LIN {X 0,Y 530.487,Z 752.804,A -85,B 0,C 180,E1 -4231.898,E2 -4231.898} C_VEL
LIN {X 0,Y 530.55,Z 749.173,A -85,B 0,C 180,E1 -4233.037,E2 -4233.037} C_VEL
LIN {X 0,Y 530.595,Z 744.443,A -85,B 0,C 180,E1 -4234.178,E2 -4234.178} C_VEL
LIN {X 0,Y 530.684,Z 738.476,A -85,B 0,C 180,E1 -4235.319,E2 -4235.319} C_VEL
LIN {X 0,Y 530.899,Z 731.608,A -85,B 0,C 180,E1 -4236.382,E2 -4236.382} C_VEL
LIN {X 0,Y 531.003,Z 723.637,A -85,B 0,C 180,E1 -4237.395,E2 -4237.395} C_VEL
LIN {X 0,Y 531.252,Z 713.214,A -85,B 0,C 180,E1 -4238.463,E2 -4238.463} C_VEL
LIN {X 0,Y 531.557,Z 702.842,A -85,B 0,C 180,E1 -4239.321,E2 -4239.321} C_VEL
LIN {X 0,Y 531.809,Z 691.176,A -85,B 0,C 180,E1 -4240.084,E2 -4240.084} C_VEL
LIN {X 0,Y 532.085,Z 678.914,A -85,B 0,C 180,E1 -4240.704,E2 -4240.704} C_VEL
LIN {X 0,Y 532.25,Z 666.678,A -85,B 0,C 180,E1 -4241.158,E2 -4241.158} C_VEL
LIN {X 0,Y 532.378,Z 652.951,A -85,B 0,C 180,E1 -4241.493,E2 -4241.493} C_VEL
LIN {X 0,Y 532.801,Z 555.086,A -85,B 0,C 180,E1 -4242.828,E2 -4242.828} C_VEL
LIN {X 0,Y 531.345,Z 546.226,A -85,B 0,C 180,E1 -4242.994,E2 -4242.994} C_VEL
LIN {X 0,Y 531.703,Z 526.604,A -85,B 0,C 180,E1 -4246.115,E2 -4246.115} C_VEL
LIN {X 0,Y 532.063,Z 506.634,A -85,B 0,C 180,E1 -4249.282,E2 -4249.282} C_VEL
LIN {X 0,Y 532.005,Z 498.624,A -85,B 0,C 180,E1 -4250.561,E2 -4250.561} C_VEL
LIN {X 0,Y 531.024,Z 493.342,A -85,B 0,C 180,E1 -4251.445,E2 -4251.445} C_VEL
LIN {X 0,Y 530.974,Z 493.345,A -85,B 0,C 180,E1 -4254.224,E2 -4254.224} C_VEL
LIN {X 0,Y 531.004,Z 493.343,A -85,B 0,C 180,E1 -4256.743,E2 -4256.743} C_VEL
LIN {X 0,Y 530.984,Z 493.345,A -85,B 0,C 180,E1 -4259.322,E2 -4259.322} C_VEL
LIN {X 0,Y 530.981,Z 493.34,A -85,B 0,C 180,E1 -4262.102,E2 -4262.102} C_VEL
LIN {X 0,Y 530.977,Z 493.347,A -85,B 0,C 180,E1 -4264.851,E2 -4264.851} C_VEL
LIN {X 0,Y 530.966,Z 493.343,A -85,B 0,C 180,E1 -4267.507,E2 -4267.507} C_VEL
LIN {X 0,Y 530.984,Z 493.34,A -85,B 0,C 180,E1 -4270.431,E2 -4270.431} C_VEL
LIN {X 0,Y 530.97,Z 493.343,A -85,B 0,C 180,E1 -4273.281,E2 -4273.281} C_VEL
LIN {X 0,Y 530.985,Z 493.336,A -85,B 0,C 180,E1 -4275.62,E2 -4275.62} C_VEL
LIN {X 0,Y 530.997,Z 493.342,A -85,B 0,C 180,E1 -4278.564,E2 -4278.564} C_VEL
LIN {X 0,Y 530.955,Z 493.343,A -85,B 0,C 180,E1 -4281.529,E2 -4281.529} C_VEL
LIN {X 0,Y 530.978,Z 493.344,A -85,B 0,C 180,E1 -4284.381,E2 -4284.381} C_VEL
LIN {X 0,Y 531.08,Z 493.373,A -85,B 0,C 180,E1 -4287.821,E2 -4287.821} C_VEL
LIN {X 0,Y 531.094,Z 499.282,A -85,B 0,C 180,E1 -4289.125,E2 -4289.125} C_VEL
LIN {X 0,Y 532.826,Z 509.254,A -85,B 0,C 180,E1 -4289.312,E2 -4289.312} C_VEL
LIN {X 0,Y 532.404,Z 603.653,A -85,B 0,C 180,E1 -4290.621,E2 -4290.621} C_VEL
LIN {X 0,Y 532.272,Z 614.13,A -85,B 0,C 180,E1 -4290.863,E2 -4290.863} C_VEL
LIN {X 0,Y 532.119,Z 623.742,A -85,B 0,C 180,E1 -4291.179,E2 -4291.179} C_VEL
LIN {X 0,Y 531.949,Z 633.546,A -85,B 0,C 180,E1 -4291.6,E2 -4291.6} C_VEL
LIN {X 0,Y 531.722,Z 643.095,A -85,B 0,C 180,E1 -4292.115,E2 -4292.115} C_VEL
LIN {X 0,Y 531.547,Z 651.225,A -85,B 0,C 180,E1 -4292.648,E2 -4292.648} C_VEL
LIN {X 0,Y 531.367,Z 659.308,A -85,B 0,C 180,E1 -4293.276,E2 -4293.276} C_VEL
LIN {X 0,Y 531.156,Z 667.23,A -85,B 0,C 180,E1 -4294.005,E2 -4294.005} C_VEL
LIN {X 0,Y 530.965,Z 673.978,A -85,B 0,C 180,E1 -4294.731,E2 -4294.731} C_VEL
LIN {X 0,Y 530.842,Z 680.541,A -85,B 0,C 180,E1 -4295.56,E2 -4295.56} C_VEL
LIN {X 0,Y 530.671,Z 687.347,A -85,B 0,C 180,E1 -4296.59,E2 -4296.59} C_VEL
LIN {X 0,Y 530.611,Z 691.992,A -85,B 0,C 180,E1 -4297.411,E2 -4297.411} C_VEL
LIN {X 0,Y 530.496,Z 697.526,A -85,B 0,C 180,E1 -4298.634,E2 -4298.634} C_VEL
LIN {X 0,Y 530.493,Z 700.569,A -85,B 0,C 180,E1 -4299.447,E2 -4299.447} C_VEL
LIN {X 0,Y 530.39,Z 703.984,A -85,B 0,C 180,E1 -4300.654,E2 -4300.654} C_VEL
LIN {X 0,Y 530.364,Z 705.668,A -85,B 0,C 180,E1 -4301.456,E2 -4301.456} C_VEL
LIN {X 0,Y 530.372,Z 707.219,A -85,B 0,C 180,E1 -4302.564,E2 -4302.564} C_VEL
LIN {X 0,Y 530.332,Z 707.983,A -85,B 0,C 180,E1 -4303.841,E2 -4303.841} C_VEL
LIN {X 0,Y 530.394,Z 707.28,A -85,B 0,C 180,E1 -4305.418,E2 -4305.418} C_VEL
LIN {X 0,Y 530.399,Z 706.401,A -85,B 0,C 180,E1 -4306.201,E2 -4306.201} C_VEL
LIN {X 0,Y 530.442,Z 703.113,A -85,B 0,C 180,E1 -4307.761,E2 -4307.761} C_VEL
LIN {X 0,Y 530.504,Z 699.364,A -85,B 0,C 180,E1 -4308.967,E2 -4308.967} C_VEL
LIN {X 0,Y 530.567,Z 694.812,A -85,B 0,C 180,E1 -4310.084,E2 -4310.084} C_VEL
LIN {X 0,Y 530.663,Z 689.94,A -85,B 0,C 180,E1 -4311.047,E2 -4311.047} C_VEL
LIN {X 0,Y 530.773,Z 684.096,A -85,B 0,C 180,E1 -4312.008,E2 -4312.008} C_VEL
LIN {X 0,Y 530.889,Z 678.366,A -85,B 0,C 180,E1 -4312.813,E2 -4312.813} C_VEL
LIN {X 0,Y 531.042,Z 672.098,A -85,B 0,C 180,E1 -4313.571,E2 -4313.571} C_VEL
LIN {X 0,Y 531.199,Z 663.996,A -85,B 0,C 180,E1 -4314.4,E2 -4314.4} C_VEL
LIN {X 0,Y 531.408,Z 655.026,A -85,B 0,C 180,E1 -4315.163,E2 -4315.163} C_VEL
LIN {X 0,Y 531.684,Z 645.483,A -85,B 0,C 180,E1 -4315.831,E2 -4315.831} C_VEL
LIN {X 0,Y 531.887,Z 635.431,A -85,B 0,C 180,E1 -4316.401,E2 -4316.401} C_VEL
LIN {X 0,Y 532.105,Z 623.614,A -85,B 0,C 180,E1 -4316.924,E2 -4316.924} C_VEL
LIN {X 0,Y 532.333,Z 609.565,A -85,B 0,C 180,E1 -4317.351,E2 -4317.351} C_VEL
LIN {X 0,Y 532.437,Z 594.602,A -85,B 0,C 180,E1 -4317.612,E2 -4317.612} C_VEL
LIN {X 0,Y 532.749,Z 508.021,A -85,B 0,C 180,E1 -4318.795,E2 -4318.795} C_VEL
LIN {X 0,Y 531.129,Z 499.354,A -85,B 0,C 180,E1 -4318.981,E2 -4318.981} C_VEL
LIN {X 0,Y 531.13,Z 493.327,A -85,B 0,C 180,E1 -4320.426,E2 -4320.426} C_VEL
LIN {X 0,Y 531.102,Z 493.331,A -85,B 0,C 180,E1 -4323.034,E2 -4323.034} C_VEL
LIN {X 0,Y 531.083,Z 493.328,A -85,B 0,C 180,E1 -4326.077,E2 -4326.077} C_VEL
LIN {X 0,Y 531.029,Z 493.341,A -85,B 0,C 180,E1 -4329.138,E2 -4329.138} C_VEL
LIN {X 0,Y 531.032,Z 493.333,A -85,B 0,C 180,E1 -4332.225,E2 -4332.225} C_VEL
LIN {X 0,Y 530.987,Z 493.346,A -85,B 0,C 180,E1 -4335.35,E2 -4335.35} C_VEL
LIN {X 0,Y 531.007,Z 493.338,A -85,B 0,C 180,E1 -4337.723,E2 -4337.723} C_VEL
LIN {X 0,Y 530.993,Z 493.343,A -85,B 0,C 180,E1 -4340.938,E2 -4340.938} C_VEL
LIN {X 0,Y 530.971,Z 493.34,A -85,B 0,C 180,E1 -4344.225,E2 -4344.225} C_VEL
LIN {X 0,Y 531.004,Z 493.339,A -85,B 0,C 180,E1 -4346.744,E2 -4346.744} C_VEL
LIN {X 0,Y 530.993,Z 493.342,A -85,B 0,C 180,E1 -4349.322,E2 -4349.322} C_VEL
LIN {X 0,Y 530.973,Z 493.338,A -85,B 0,C 180,E1 -4352.104,E2 -4352.104} C_VEL
LIN {X 0,Y 530.985,Z 493.343,A -85,B 0,C 180,E1 -4354.855,E2 -4354.855} C_VEL
LIN {X 0,Y 530.96,Z 493.344,A -85,B 0,C 180,E1 -4357.508,E2 -4357.508} C_VEL
LIN {X 0,Y 530.979,Z 493.341,A -85,B 0,C 180,E1 -4360.433,E2 -4360.433} C_VEL
LIN {X 0,Y 530.961,Z 493.346,A -85,B 0,C 180,E1 -4363.282,E2 -4363.282} C_VEL
LIN {X 0,Y 530.983,Z 493.341,A -85,B 0,C 180,E1 -4365.622,E2 -4365.622} C_VEL
LIN {X 0,Y 530.997,Z 493.342,A -85,B 0,C 180,E1 -4368.566,E2 -4368.566} C_VEL
LIN {X 0,Y 530.957,Z 493.344,A -85,B 0,C 180,E1 -4371.53,E2 -4371.53} C_VEL
LIN {X 0,Y 530.974,Z 493.343,A -85,B 0,C 180,E1 -4374.382,E2 -4374.382} C_VEL
LIN {X 0,Y 530.97,Z 493.349,A -85,B 0,C 180,E1 -4377.134,E2 -4377.134} C_VEL
LIN {X 0,Y 530.969,Z 493.344,A -85,B 0,C 180,E1 -4379.804,E2 -4379.804} C_VEL
LIN {X 0,Y 531.015,Z 493.342,A -85,B 0,C 180,E1 -4382.468,E2 -4382.468} C_VEL
LIN {X 0,Y 531.024,Z 493.423,A -85,B 0,C 180,E1 -4383.972,E2 -4383.972} C_VEL
LIN {X 0,Y 532.778,Z 502.655,A -85,B 0,C 180,E1 -4385.336,E2 -4385.336} C_VEL
LIN {X 0,Y 532.4,Z 522.848,A -85,B 0,C 180,E1 -4388.105,E2 -4388.105} C_VEL
LIN {X 0,Y 531.968,Z 545.102,A -85,B 0,C 180,E1 -4391.115,E2 -4391.115} C_VEL
LIN {X 0,Y 531.558,Z 568.799,A -85,B 0,C 180,E1 -4394.274,E2 -4394.274} C_VEL
LIN {X 0,Y 531.509,Z 574.595,A -85,B 0,C 180,E1 -4395.044,E2 -4395.044} C_VEL
LIN {X 0,Y 532.809,Z 584.953,A -85,B 0,C 180,E1 -4395.225,E2 -4395.225} C_VEL
LIN {X 0,Y 532.437,Z 683.8,A -85,B 0,C 180,E1 -4396.572,E2 -4396.572} C_VEL
LIN {X 0,Y 532.218,Z 697.173,A -85,B 0,C 180,E1 -4396.906,E2 -4396.906} C_VEL
LIN {X 0,Y 532,Z 709.367,A -85,B 0,C 180,E1 -4397.362,E2 -4397.362} C_VEL
LIN {X 0,Y 531.806,Z 721.308,A -85,B 0,C 180,E1 -4397.967,E2 -4397.967} C_VEL
LIN {X 0,Y 531.518,Z 733.197,A -85,B 0,C 180,E1 -4398.754,E2 -4398.754} C_VEL
LIN {X 0,Y 531.251,Z 743.606,A -85,B 0,C 180,E1 -4399.616,E2 -4399.616} C_VEL
LIN {X 0,Y 531.06,Z 752.116,A -85,B 0,C 180,E1 -4400.478,E2 -4400.478} C_VEL
LIN {X 0,Y 530.886,Z 759.962,A -85,B 0,C 180,E1 -4401.435,E2 -4401.435} C_VEL
LIN {X 0,Y 530.684,Z 767.623,A -85,B 0,C 180,E1 -4402.581,E2 -4402.581} C_VEL
LIN {X 0,Y 530.604,Z 774.679,A -85,B 0,C 180,E1 -4403.918,E2 -4403.918} C_VEL
LIN {X 0,Y 530.459,Z 779.372,A -85,B 0,C 180,E1 -4405.06,E2 -4405.06} C_VEL
LIN {X 0,Y 530.516,Z 782.961,A -85,B 0,C 180,E1 -4406.202,E2 -4406.202} C_VEL
LIN {X 0,Y 530.457,Z 784.81,A -85,B 0,C 180,E1 -4406.962,E2 -4406.962} C_VEL
LIN {X 0,Y 530.41,Z 786.196,A -85,B 0,C 180,E1 -4407.722,E2 -4407.722} C_VEL
LIN {X 0,Y 530.344,Z 787.786,A -85,B 0,C 180,E1 -4409.241,E2 -4409.241} C_VEL
LIN {X 0,Y 530.342,Z 788,A -85,B 0,C 180,E1 -4410,E2 -4410} C_VEL
LIN {X 0,Y 530.361,Z 787.182,A -85,B 0,C 180,E1 -4411.519,E2 -4411.519} C_VEL
LIN {X 0,Y 530.41,Z 786.194,A -85,B 0,C 180,E1 -4412.278,E2 -4412.278} C_VEL
LIN {X 0,Y 530.457,Z 784.807,A -85,B 0,C 180,E1 -4413.038,E2 -4413.038} C_VEL
LIN {X 0,Y 530.522,Z 781.895,A -85,B 0,C 180,E1 -4414.178,E2 -4414.178} C_VEL
LIN {X 0,Y 530.525,Z 777.95,A -85,B 0,C 180,E1 -4415.321,E2 -4415.321} C_VEL
LIN {X 0,Y 530.599,Z 772.263,A -85,B 0,C 180,E1 -4416.582,E2 -4416.582} C_VEL
LIN {X 0,Y 530.758,Z 765.236,A -85,B 0,C 180,E1 -4417.8,E2 -4417.8} C_VEL
LIN {X 0,Y 530.93,Z 756.994,A -85,B 0,C 180,E1 -4418.948,E2 -4418.948} C_VEL
LIN {X 0,Y 531.137,Z 748.542,A -85,B 0,C 180,E1 -4419.905,E2 -4419.905} C_VEL
LIN {X 0,Y 531.407,Z 738.094,A -85,B 0,C 180,E1 -4420.863,E2 -4420.863} C_VEL
LIN {X 0,Y 531.646,Z 727.135,A -85,B 0,C 180,E1 -4421.672,E2 -4421.672} C_VEL
LIN {X 0,Y 531.933,Z 716.411,A -85,B 0,C 180,E1 -4422.301,E2 -4422.301} C_VEL
LIN {X 0,Y 532.124,Z 704.776,A -85,B 0,C 180,E1 -4422.829,E2 -4422.829} C_VEL
LIN {X 0,Y 532.287,Z 692.194,A -85,B 0,C 180,E1 -4423.238,E2 -4423.238} C_VEL
LIN {X 0,Y 532.462,Z 679.427,A -85,B 0,C 180,E1 -4423.5,E2 -4423.5} C_VEL
LIN {X 0,Y 532.763,Z 583.331,A -85,B 0,C 180,E1 -4424.801,E2 -4424.801} C_VEL
LIN {X 0,Y 531.493,Z 574.705,A -85,B 0,C 180,E1 -4424.96,E2 -4424.96} C_VEL
LIN {X 0,Y 531.885,Z 550.961,A -85,B 0,C 180,E1 -4428.153,E2 -4428.153} C_VEL
LIN {X 0,Y 532.418,Z 527.933,A -85,B 0,C 180,E1 -4431.284,E2 -4431.284} C_VEL
LIN {X 0,Y 532.874,Z 507.288,A -85,B 0,C 180,E1 -4434.132,E2 -4434.132} C_VEL
LIN {X 0,Y 532.831,Z 502.44,A -85,B 0,C 180,E1 -4434.822,E2 -4434.822} C_VEL
LIN {X 0,Y 531.018,Z 493.34,A -85,B 0,C 180,E1 -4436.231,E2 -4436.231} C_VEL
LIN {X 0,Y 530.988,Z 493.347,A -85,B 0,C 180,E1 -4439.125,E2 -4439.125} C_VEL
LIN {X 0,Y 530.974,Z 493.341,A -85,B 0,C 180,E1 -4442.101,E2 -4442.101} C_VEL
LIN {X 0,Y 530.97,Z 493.345,A -85,B 0,C 180,E1 -4444.851,E2 -4444.851} C_VEL
LIN {X 0,Y 530.963,Z 493.336,A -85,B 0,C 180,E1 -4447.507,E2 -4447.507} C_VEL
LIN {X 0,Y 530.981,Z 493.338,A -85,B 0,C 180,E1 -4450.432,E2 -4450.432} C_VEL
LIN {X 0,Y 530.966,Z 493.346,A -85,B 0,C 180,E1 -4453.281,E2 -4453.281} C_VEL
LIN {X 0,Y 530.983,Z 493.342,A -85,B 0,C 180,E1 -4455.62,E2 -4455.62} C_VEL
LIN {X 0,Y 531.001,Z 493.335,A -85,B 0,C 180,E1 -4458.565,E2 -4458.565} C_VEL
LIN {X 0,Y 530.953,Z 493.345,A -85,B 0,C 180,E1 -4461.529,E2 -4461.529} C_VEL
LIN {X 0,Y 530.976,Z 493.337,A -85,B 0,C 180,E1 -4464.382,E2 -4464.382} C_VEL
LIN {X 0,Y 530.968,Z 493.349,A -85,B 0,C 180,E1 -4467.133,E2 -4467.133} C_VEL
LIN {X 0,Y 530.978,Z 493.337,A -85,B 0,C 180,E1 -4469.804,E2 -4469.804} C_VEL
LIN {X 0,Y 531.009,Z 493.336,A -85,B 0,C 180,E1 -4472.466,E2 -4472.466} C_VEL
LIN {X 0,Y 530.999,Z 493.341,A -85,B 0,C 180,E1 -4474.942,E2 -4474.942} C_VEL
LIN {X 0,Y 530.963,Z 493.34,A -85,B 0,C 180,E1 -4478.246,E2 -4478.246} C_VEL
LIN {X 0,Y 530.988,Z 493.34,A -85,B 0,C 180,E1 -4480.677,E2 -4480.677} C_VEL
LIN {X 0,Y 530.984,Z 493.341,A -85,B 0,C 180,E1 -4483.071,E2 -4483.071} C_VEL
LIN {X 0,Y 531.009,Z 493.339,A -85,B 0,C 180,E1 -4485.436,E2 -4485.436} C_VEL
LIN {X 0,Y 531.042,Z 493.333,A -85,B 0,C 180,E1 -4488.55,E2 -4488.55} C_VEL
LIN {X 0,Y 531.051,Z 493.326,A -85,B 0,C 180,E1 -4491.63,E2 -4491.63} C_VEL
LIN {X 0,Y 531.135,Z 493.321,A -85,B 0,C 180,E1 -4494.686,E2 -4494.686} C_VEL
LIN {X 0,Y 531.13,Z 493.319,A -85,B 0,C 180,E1 -4497.725,E2 -4497.725} C_VEL
LIN {X 0,Y 531.148,Z 493.314,A -85,B 0,C 180,E1 -4500.758,E2 -4500.758} C_VEL
LIN {X 0,Y 531.103,Z 493.33,A -85,B 0,C 180,E1 -4503.034,E2 -4503.034} C_VEL
LIN {X 0,Y 531.083,Z 493.324,A -85,B 0,C 180,E1 -4506.077,E2 -4506.077} C_VEL
LIN {X 0,Y 531.028,Z 493.335,A -85,B 0,C 180,E1 -4509.138,E2 -4509.138} C_VEL
LIN {X 0,Y 531.032,Z 493.332,A -85,B 0,C 180,E1 -4512.225,E2 -4512.225} C_VEL
LIN {X 0,Y 530.988,Z 493.336,A -85,B 0,C 180,E1 -4515.35,E2 -4515.35} C_VEL
LIN {X 0,Y 530.989,Z 493.338,A -85,B 0,C 180,E1 -4518.522,E2 -4518.522} C_VEL
LIN {X 0,Y 530.994,Z 493.345,A -85,B 0,C 180,E1 -4520.938,E2 -4520.938} C_VEL
LIN {X 0,Y 530.972,Z 493.336,A -85,B 0,C 180,E1 -4524.225,E2 -4524.225} C_VEL
LIN {X 0,Y 531.006,Z 493.34,A -85,B 0,C 180,E1 -4526.744,E2 -4526.744} C_VEL
LIN {X 0,Y 530.994,Z 493.339,A -85,B 0,C 180,E1 -4529.322,E2 -4529.322} C_VEL
LIN {X 0,Y 530.974,Z 493.34,A -85,B 0,C 180,E1 -4532.104,E2 -4532.104} C_VEL
LIN {X 0,Y 530.987,Z 493.343,A -85,B 0,C 180,E1 -4534.856,E2 -4534.856} C_VEL
LIN {X 0,Y 530.97,Z 493.343,A -85,B 0,C 180,E1 -4537.508,E2 -4537.508} C_VEL
LIN {X 0,Y 530.981,Z 493.34,A -85,B 0,C 180,E1 -4540.433,E2 -4540.433} C_VEL
LIN {X 0,Y 530.963,Z 493.346,A -85,B 0,C 180,E1 -4543.283,E2 -4543.283} C_VEL
LIN {X 0,Y 530.955,Z 493.343,A -85,B 0,C 180,E1 -4543.578,E2 -4543.578} C_VEL
LIN {X 0,Y 530.285,Z 493.426,A -85,B 0,C 180,E1 -4544.212,E2 -4544.212} C_VEL
LIN {X 0,Y 527.441,Z 493.786,A -85,B 0,C 180,E1 -4545.241,E2 -4545.241} C_VEL
LIN {X 0,Y 525.039,Z 494.089,A -85,B 0,C 180,E1 -4546.069,E2 -4546.069} C_VEL
LIN {X 0,Y 524.007,Z 494.216,A -85,B 0,C 180,E1 -4546.709,E2 -4546.709} C_VEL
LIN {X 0,Y 523.922,Z 494.224,A -85,B 0,C 180,E1 -4546.925,E2 -4546.925} C_VEL
LIN {X 0,Y 523.947,Z 494.215,A -85,B 0,C 180,E1 -4549.922,E2 -4549.922} C_VEL
LIN {X 0,Y 523.907,Z 494.227,A -85,B 0,C 180,E1 -4552.869,E2 -4552.869} C_VEL
LIN {X 0,Y 523.933,Z 494.218,A -85,B 0,C 180,E1 -4555.711,E2 -4555.711} C_VEL
LIN {X 0,Y 523.922,Z 494.218,A -85,B 0,C 180,E1 -4558.457,E2 -4558.457} C_VEL
LIN {X 0,Y 523.941,Z 494.224,A -85,B 0,C 180,E1 -4561.126,E2 -4561.126} C_VEL
LIN {X 0,Y 523.99,Z 494.215,A -85,B 0,C 180,E1 -4564.226,E2 -4564.226} C_VEL
LIN {X 0,Y 524.037,Z 494.411,A -85,B 0,C 180,E1 -4564.542,E2 -4564.542} C_VEL
LIN {X 0,Y 525.161,Z 501.036,A -85,B 0,C 180,E1 -4565.65,E2 -4565.65} C_VEL
LIN {X 0,Y 524.955,Z 515.568,A -85,B 0,C 180,E1 -4567.985,E2 -4567.985} C_VEL
LIN {X 0,Y 524.609,Z 533.464,A -85,B 0,C 180,E1 -4570.84,E2 -4570.84} C_VEL
LIN {X 0,Y 524.393,Z 546.374,A -85,B 0,C 180,E1 -4572.896,E2 -4572.896} C_VEL
LIN {X 0,Y 525.949,Z 556.228,A -85,B 0,C 180,E1 -4573.079,E2 -4573.079} C_VEL
LIN {X 0,Y 525.506,Z 654.053,A -85,B 0,C 180,E1 -4574.437,E2 -4574.437} C_VEL
LIN {X 0,Y 525.36,Z 666.776,A -85,B 0,C 180,E1 -4574.755,E2 -4574.755} C_VEL
LIN {X 0,Y 525.163,Z 679.178,A -85,B 0,C 180,E1 -4575.221,E2 -4575.221} C_VEL
LIN {X 0,Y 524.87,Z 691.551,A -85,B 0,C 180,E1 -4575.856,E2 -4575.856} C_VEL
LIN {X 0,Y 524.55,Z 703.291,A -85,B 0,C 180,E1 -4576.637,E2 -4576.637} C_VEL
LIN {X 0,Y 524.254,Z 713.693,A -85,B 0,C 180,E1 -4577.516,E2 -4577.516} C_VEL
LIN {X 0,Y 523.958,Z 723.948,A -85,B 0,C 180,E1 -4578.589,E2 -4578.589} C_VEL
LIN {X 0,Y 523.78,Z 732.813,A -85,B 0,C 180,E1 -4579.759,E2 -4579.759} C_VEL
LIN {X 0,Y 523.605,Z 739.95,A -85,B 0,C 180,E1 -4580.926,E2 -4580.926} C_VEL
LIN {X 0,Y 523.475,Z 746.472,A -85,B 0,C 180,E1 -4582.285,E2 -4582.285} C_VEL
LIN {X 0,Y 523.438,Z 750.931,A -85,B 0,C 180,E1 -4583.503,E2 -4583.503} C_VEL
LIN {X 0,Y 523.389,Z 753.986,A -85,B 0,C 180,E1 -4584.607,E2 -4584.607} C_VEL
LIN {X 0,Y 523.384,Z 756.79,A -85,B 0,C 180,E1 -4586.15,E2 -4586.15} C_VEL
LIN {X 0,Y 523.36,Z 757.567,A -85,B 0,C 180,E1 -4586.921,E2 -4586.921} C_VEL
LIN {X 0,Y 523.334,Z 757.934,A -85,B 0,C 180,E1 -4587.691,E2 -4587.691} C_VEL
LIN {X 0,Y 523.25,Z 757.528,A -85,B 0,C 180,E1 -4589.23,E2 -4589.23} C_VEL
LIN {X 0,Y 523.249,Z 756.705,A -85,B 0,C 180,E1 -4590,E2 -4590} C_VEL
LIN {X 0,Y 523.305,Z 753.862,A -85,B 0,C 180,E1 -4591.539,E2 -4591.539} C_VEL
LIN {X 0,Y 523.422,Z 750.597,A -85,B 0,C 180,E1 -4592.694,E2 -4592.694} C_VEL
LIN {X 0,Y 523.497,Z 746.295,A -85,B 0,C 180,E1 -4593.849,E2 -4593.849} C_VEL
LIN {X 0,Y 523.635,Z 739.763,A -85,B 0,C 180,E1 -4595.198,E2 -4595.198} C_VEL
LIN {X 0,Y 523.829,Z 732.285,A -85,B 0,C 180,E1 -4596.409,E2 -4596.409} C_VEL
LIN {X 0,Y 523.975,Z 723.823,A -85,B 0,C 180,E1 -4597.514,E2 -4597.514} C_VEL
LIN {X 0,Y 524.259,Z 713.652,A -85,B 0,C 180,E1 -4598.577,E2 -4598.577} C_VEL
LIN {X 0,Y 524.579,Z 703.366,A -85,B 0,C 180,E1 -4599.446,E2 -4599.446} C_VEL
LIN {X 0,Y 524.825,Z 693.456,A -85,B 0,C 180,E1 -4600.123,E2 -4600.123} C_VEL
LIN {X 0,Y 525.08,Z 681.754,A -85,B 0,C 180,E1 -4600.751,E2 -4600.751} C_VEL
LIN {X 0,Y 525.341,Z 668.431,A -85,B 0,C 180,E1 -4601.283,E2 -4601.283} C_VEL
LIN {X 0,Y 525.484,Z 655.682,A -85,B 0,C 180,E1 -4601.622,E2 -4601.622} C_VEL
LIN {X 0,Y 525.666,Z 625.753,A -85,B 0,C 180,E1 -4602.058,E2 -4602.058} C_VEL
LIN {X 0,Y 525.821,Z 554.936,A -85,B 0,C 180,E1 -4603.032,E2 -4603.032} C_VEL
LIN {X 0,Y 524.35,Z 546.179,A -85,B 0,C 180,E1 -4603.22,E2 -4603.22} C_VEL
LIN {X 0,Y 524.718,Z 527.974,A -85,B 0,C 180,E1 -4606.136,E2 -4606.136} C_VEL
LIN {X 0,Y 525.07,Z 509.153,A -85,B 0,C 180,E1 -4609.143,E2 -4609.143} C_VEL
LIN {X 0,Y 525.17,Z 500.793,A -85,B 0,C 180,E1 -4610.484,E2 -4610.484} C_VEL
LIN {X 0,Y 523.966,Z 494.22,A -85,B 0,C 180,E1 -4611.593,E2 -4611.593} C_VEL
LIN {X 0,Y 523.935,Z 494.225,A -85,B 0,C 180,E1 -4614.571,E2 -4614.571} C_VEL
LIN {X 0,Y 523.953,Z 494.222,A -85,B 0,C 180,E1 -4617.132,E2 -4617.132} C_VEL
LIN {X 0,Y 523.944,Z 494.218,A -85,B 0,C 180,E1 -4619.755,E2 -4619.755} C_VEL
LIN {X 0,Y 523.941,Z 494.219,A -85,B 0,C 180,E1 -4622.448,E2 -4622.448} C_VEL
LIN {X 0,Y 523.923,Z 494.223,A -85,B 0,C 180,E1 -4625.226,E2 -4625.226} C_VEL
LIN {X 0,Y 523.917,Z 494.219,A -85,B 0,C 180,E1 -4628.101,E2 -4628.101} C_VEL
LIN {X 0,Y 523.961,Z 494.217,A -85,B 0,C 180,E1 -4631.31,E2 -4631.31} C_VEL
LIN {X 0,Y 523.954,Z 494.22,A -85,B 0,C 180,E1 -4634.69,E2 -4634.69} C_VEL
LIN {X 0,Y 523.954,Z 494.214,A -85,B 0,C 180,E1 -4637.881,E2 -4637.881} C_VEL
LIN {X 0,Y 523.92,Z 494.226,A -85,B 0,C 180,E1 -4640.915,E2 -4640.915} C_VEL
LIN {X 0,Y 523.924,Z 494.219,A -85,B 0,C 180,E1 -4643.827,E2 -4643.827} C_VEL
LIN {X 0,Y 523.944,Z 494.224,A -85,B 0,C 180,E1 -4646.635,E2 -4646.635} C_VEL
LIN {X 0,Y 524.044,Z 494.323,A -85,B 0,C 180,E1 -4647.737,E2 -4647.737} C_VEL
LIN {X 0,Y 524.099,Z 499.432,A -85,B 0,C 180,E1 -4648.908,E2 -4648.908} C_VEL
LIN {X 0,Y 525.991,Z 510.041,A -85,B 0,C 180,E1 -4649.122,E2 -4649.122} C_VEL
LIN {X 0,Y 525.502,Z 605.175,A -85,B 0,C 180,E1 -4650.472,E2 -4650.472} C_VEL
LIN {X 0,Y 525.337,Z 617.655,A -85,B 0,C 180,E1 -4650.784,E2 -4650.784} C_VEL
LIN {X 0,Y 525.095,Z 631.166,A -85,B 0,C 180,E1 -4651.304,E2 -4651.304} C_VEL
LIN {X 0,Y 524.858,Z 641.419,A -85,B 0,C 180,E1 -4651.835,E2 -4651.835} C_VEL
LIN {X 0,Y 524.622,Z 651.262,A -85,B 0,C 180,E1 -4652.472,E2 -4652.472} C_VEL
LIN {X 0,Y 524.362,Z 660.618,A -85,B 0,C 180,E1 -4653.213,E2 -4653.213} C_VEL
LIN {X 0,Y 524.155,Z 669.157,A -85,B 0,C 180,E1 -4654.029,E2 -4654.029} C_VEL
LIN {X 0,Y 523.916,Z 675.913,A -85,B 0,C 180,E1 -4654.792,E2 -4654.792} C_VEL
LIN {X 0,Y 523.777,Z 682.572,A -85,B 0,C 180,E1 -4655.679,E2 -4655.679} C_VEL
LIN {X 0,Y 523.613,Z 688.825,A -85,B 0,C 180,E1 -4656.674,E2 -4656.674} C_VEL
LIN {X 0,Y 523.551,Z 693.427,A -85,B 0,C 180,E1 -4657.548,E2 -4657.548} C_VEL
LIN {X 0,Y 523.412,Z 698.536,A -85,B 0,C 180,E1 -4658.744,E2 -4658.744} C_VEL
LIN {X 0,Y 523.377,Z 702.754,A -85,B 0,C 180,E1 -4660.043,E2 -4660.043} C_VEL
LIN {X 0,Y 523.268,Z 705.436,A -85,B 0,C 180,E1 -4661.195,E2 -4661.195} C_VEL
LIN {X 0,Y 523.279,Z 707.688,A -85,B 0,C 180,E1 -4662.814,E2 -4662.814} C_VEL
LIN {X 0,Y 523.232,Z 708.09,A -85,B 0,C 180,E1 -4663.616,E2 -4663.616} C_VEL
LIN {X 0,Y 523.295,Z 707.706,A -85,B 0,C 180,E1 -4665.23,E2 -4665.23} C_VEL
LIN {X 0,Y 523.295,Z 706.9,A -85,B 0,C 180,E1 -4666.01,E2 -4666.01} C_VEL
LIN {X 0,Y 523.358,Z 703.965,A -85,B 0,C 180,E1 -4667.593,E2 -4667.593} C_VEL
LIN {X 0,Y 523.439,Z 700.276,A -85,B 0,C 180,E1 -4668.866,E2 -4668.866} C_VEL
LIN {X 0,Y 523.496,Z 696.156,A -85,B 0,C 180,E1 -4669.949,E2 -4669.949} C_VEL
LIN {X 0,Y 523.614,Z 690.511,A -85,B 0,C 180,E1 -4671.12,E2 -4671.12} C_VEL
LIN {X 0,Y 523.798,Z 683.493,A -85,B 0,C 180,E1 -4672.289,E2 -4672.289} C_VEL
LIN {X 0,Y 524.028,Z 674.116,A -85,B 0,C 180,E1 -4673.529,E2 -4673.529} C_VEL
LIN {X 0,Y 524.231,Z 664.67,A -85,B 0,C 180,E1 -4674.519,E2 -4674.519} C_VEL
LIN {X 0,Y 524.453,Z 655.716,A -85,B 0,C 180,E1 -4675.292,E2 -4675.292} C_VEL
LIN {X 0,Y 524.742,Z 646.192,A -85,B 0,C 180,E1 -4675.968,E2 -4675.968} C_VEL
LIN {X 0,Y 524.95,Z 636.168,A -85,B 0,C 180,E1 -4676.546,E2 -4676.546} C_VEL
LIN {X 0,Y 525.191,Z 624.351,A -85,B 0,C 180,E1 -4677.075,E2 -4677.075} C_VEL
LIN {X 0,Y 525.417,Z 610.4,A -85,B 0,C 180,E1 -4677.508,E2 -4677.508} C_VEL
LIN {X 0,Y 525.53,Z 595.603,A -85,B 0,C 180,E1 -4677.772,E2 -4677.772} C_VEL
LIN {X 0,Y 525.904,Z 508.958,A -85,B 0,C 180,E1 -4678.983,E2 -4678.983} C_VEL
LIN {X 0,Y 524.164,Z 499.964,A -85,B 0,C 180,E1 -4679.184,E2 -4679.184} C_VEL
LIN {X 0,Y 524.111,Z 494.202,A -85,B 0,C 180,E1 -4680.576,E2 -4680.576} C_VEL
LIN {X 0,Y 524.069,Z 494.207,A -85,B 0,C 180,E1 -4683.075,E2 -4683.075} C_VEL
LIN {X 0,Y 524.044,Z 494.205,A -85,B 0,C 180,E1 -4686.159,E2 -4686.159} C_VEL
LIN {X 0,Y 523.996,Z 494.218,A -85,B 0,C 180,E1 -4689.262,E2 -4689.262} C_VEL
LIN {X 0,Y 524.014,Z 494.21,A -85,B 0,C 180,E1 -4691.751,E2 -4691.751} C_VEL
LIN {X 0,Y 523.982,Z 494.218,A -85,B 0,C 180,E1 -4695.053,E2 -4695.053} C_VEL
LIN {X 0,Y 523.955,Z 494.215,A -85,B 0,C 180,E1 -4697.969,E2 -4697.969} C_VEL
LIN {X 0,Y 523.963,Z 494.214,A -85,B 0,C 180,E1 -4700.41,E2 -4700.41} C_VEL
LIN {X 0,Y 523.908,Z 494.225,A -85,B 0,C 180,E1 -4702.894,E2 -4702.894} C_VEL
LIN {X 0,Y 523.947,Z 494.22,A -85,B 0,C 180,E1 -4705.419,E2 -4705.419} C_VEL
LIN {X 0,Y 523.963,Z 494.212,A -85,B 0,C 180,E1 -4707.999,E2 -4707.999} C_VEL
LIN {X 0,Y 523.945,Z 494.219,A -85,B 0,C 180,E1 -4710.857,E2 -4710.857} C_VEL
LIN {X 0,Y 523.956,Z 494.214,A -85,B 0,C 180,E1 -4713.736,E2 -4713.736} C_VEL
LIN {X 0,Y 523.916,Z 494.219,A -85,B 0,C 180,E1 -4716.405,E2 -4716.405} C_VEL
LIN {X 0,Y 523.919,Z 494.227,A -85,B 0,C 180,E1 -4719.085,E2 -4719.085} C_VEL
LIN {X 0,Y 523.951,Z 494.215,A -85,B 0,C 180,E1 -4722.119,E2 -4722.119} C_VEL
LIN {X 0,Y 523.951,Z 494.22,A -85,B 0,C 180,E1 -4725.309,E2 -4725.309} C_VEL
LIN {X 0,Y 523.958,Z 494.221,A -85,B 0,C 180,E1 -4728.69,E2 -4728.69} C_VEL
LIN {X 0,Y 523.914,Z 494.22,A -85,B 0,C 180,E1 -4731.899,E2 -4731.899} C_VEL
LIN {X 0,Y 523.932,Z 494.226,A -85,B 0,C 180,E1 -4734.91,E2 -4734.91} C_VEL
LIN {X 0,Y 523.941,Z 494.22,A -85,B 0,C 180,E1 -4737.679,E2 -4737.679} C_VEL
LIN {X 0,Y 523.954,Z 494.223,A -85,B 0,C 180,E1 -4740.677,E2 -4740.677} C_VEL
LIN {X 0,Y 523.98,Z 494.218,A -85,B 0,C 180,E1 -4743.73,E2 -4743.73} C_VEL
LIN {X 0,Y 523.994,Z 494.33,A -85,B 0,C 180,E1 -4743.811,E2 -4743.811} C_VEL
LIN {X 0,Y 525.864,Z 504.528,A -85,B 0,C 180,E1 -4745.34,E2 -4745.34} C_VEL
LIN {X 0,Y 525.333,Z 526.658,A -85,B 0,C 180,E1 -4748.414,E2 -4748.414} C_VEL
LIN {X 0,Y 524.9,Z 547.416,A -85,B 0,C 180,E1 -4751.256,E2 -4751.256} C_VEL
LIN {X 0,Y 524.49,Z 571.106,A -85,B 0,C 180,E1 -4754.455,E2 -4754.455} C_VEL
LIN {X 0,Y 524.44,Z 573.938,A -85,B 0,C 180,E1 -4754.837,E2 -4754.837} C_VEL
LIN {X 0,Y 525.929,Z 585.432,A -85,B 0,C 180,E1 -4755.052,E2 -4755.052} C_VEL
LIN {X 0,Y 525.506,Z 683.603,A -85,B 0,C 180,E1 -4756.416,E2 -4756.416} C_VEL
LIN {X 0,Y 525.26,Z 696.831,A -85,B 0,C 180,E1 -4756.754,E2 -4756.754} C_VEL
LIN {X 0,Y 525.006,Z 709.598,A -85,B 0,C 180,E1 -4757.24,E2 -4757.24} C_VEL
LIN {X 0,Y 524.789,Z 721.493,A -85,B 0,C 180,E1 -4757.856,E2 -4757.856} C_VEL
LIN {X 0,Y 524.514,Z 732.72,A -85,B 0,C 180,E1 -4758.602,E2 -4758.602} C_VEL
LIN {X 0,Y 524.223,Z 743.297,A -85,B 0,C 180,E1 -4759.475,E2 -4759.475} C_VEL
LIN {X 0,Y 524.026,Z 751.947,A -85,B 0,C 180,E1 -4760.349,E2 -4760.349} C_VEL
LIN {X 0,Y 523.851,Z 759.917,A -85,B 0,C 180,E1 -4761.319,E2 -4761.319} C_VEL
LIN {X 0,Y 523.633,Z 767.623,A -85,B 0,C 180,E1 -4762.481,E2 -4762.481} C_VEL
LIN {X 0,Y 523.515,Z 774.679,A -85,B 0,C 180,E1 -4763.835,E2 -4763.835} C_VEL
LIN {X 0,Y 523.384,Z 779.372,A -85,B 0,C 180,E1 -4764.993,E2 -4764.993} C_VEL
LIN {X 0,Y 523.443,Z 782.96,A -85,B 0,C 180,E1 -4766.151,E2 -4766.151} C_VEL
LIN {X 0,Y 523.367,Z 784.81,A -85,B 0,C 180,E1 -4766.921,E2 -4766.921} C_VEL
LIN {X 0,Y 523.334,Z 786.196,A -85,B 0,C 180,E1 -4767.691,E2 -4767.691} C_VEL
LIN {X 0,Y 523.25,Z 787.786,A -85,B 0,C 180,E1 -4769.23,E2 -4769.23} C_VEL
LIN {X 0,Y 523.246,Z 788,A -85,B 0,C 180,E1 -4770,E2 -4770} C_VEL
LIN {X 0,Y 523.274,Z 787.182,A -85,B 0,C 180,E1 -4771.539,E2 -4771.539} C_VEL
LIN {X 0,Y 523.334,Z 786.193,A -85,B 0,C 180,E1 -4772.309,E2 -4772.309} C_VEL
LIN {X 0,Y 523.367,Z 784.807,A -85,B 0,C 180,E1 -4773.079,E2 -4773.079} C_VEL
LIN {X 0,Y 523.441,Z 781.894,A -85,B 0,C 180,E1 -4774.235,E2 -4774.235} C_VEL
LIN {X 0,Y 523.464,Z 777.95,A -85,B 0,C 180,E1 -4775.393,E2 -4775.393} C_VEL
LIN {X 0,Y 523.523,Z 772.727,A -85,B 0,C 180,E1 -4776.581,E2 -4776.581} C_VEL
LIN {X 0,Y 523.664,Z 766.465,A -85,B 0,C 180,E1 -4777.713,E2 -4777.713} C_VEL
LIN {X 0,Y 523.852,Z 758.413,A -85,B 0,C 180,E1 -4778.875,E2 -4778.875} C_VEL
LIN {X 0,Y 524.077,Z 750.157,A -85,B 0,C 180,E1 -4779.845,E2 -4779.845} C_VEL
LIN {X 0,Y 524.321,Z 740.083,A -85,B 0,C 180,E1 -4780.816,E2 -4780.816} C_VEL
LIN {X 0,Y 524.588,Z 730.144,A -85,B 0,C 180,E1 -4781.593,E2 -4781.593} C_VEL
LIN {X 0,Y 524.857,Z 718.586,A -85,B 0,C 180,E1 -4782.314,E2 -4782.314} C_VEL
LIN {X 0,Y 525.103,Z 706.346,A -85,B 0,C 180,E1 -4782.905,E2 -4782.905} C_VEL
LIN {X 0,Y 525.295,Z 693.952,A -85,B 0,C 180,E1 -4783.343,E2 -4783.343} C_VEL
LIN {X 0,Y 525.508,Z 681.189,A -85,B 0,C 180,E1 -4783.633,E2 -4783.633} C_VEL
LIN {X 0,Y 525.854,Z 583.792,A -85,B 0,C 180,E1 -4784.98,E2 -4784.98} C_VEL
LIN {X 0,Y 524.479,Z 574.256,A -85,B 0,C 180,E1 -4785.165,E2 -4785.165} C_VEL
LIN {X 0,Y 524.922,Z 550.986,A -85,B 0,C 180,E1 -4788.342,E2 -4788.342} C_VEL
LIN {X 0,Y 525.492,Z 527.511,A -85,B 0,C 180,E1 -4791.579,E2 -4791.579} C_VEL
LIN {X 0,Y 526.001,Z 506.907,A -85,B 0,C 180,E1 -4794.468,E2 -4794.468} C_VEL
LIN {X 0,Y 525.646,Z 502.315,A -85,B 0,C 180,E1 -4795.146,E2 -4795.146} C_VEL
LIN {X 0,Y 523.959,Z 494.219,A -85,B 0,C 180,E1 -4796.432,E2 -4796.432} C_VEL
LIN {X 0,Y 523.954,Z 494.223,A -85,B 0,C 180,E1 -4799.323,E2 -4799.323} C_VEL
LIN {X 0,Y 523.938,Z 494.217,A -85,B 0,C 180,E1 -4802.32,E2 -4802.32} C_VEL
LIN {X 0,Y 523.919,Z 494.227,A -85,B 0,C 180,E1 -4805.226,E2 -4805.226} C_VEL
LIN {X 0,Y 523.914,Z 494.208,A -85,B 0,C 180,E1 -4808.101,E2 -4808.101} C_VEL
LIN {X 0,Y 523.958,Z 494.222,A -85,B 0,C 180,E1 -4811.31,E2 -4811.31} C_VEL
LIN {X 0,Y 523.951,Z 494.215,A -85,B 0,C 180,E1 -4814.691,E2 -4814.691} C_VEL
LIN {X 0,Y 523.951,Z 494.212,A -85,B 0,C 180,E1 -4817.881,E2 -4817.881} C_VEL
LIN {X 0,Y 523.918,Z 494.224,A -85,B 0,C 180,E1 -4820.915,E2 -4820.915} C_VEL
LIN {X 0,Y 523.921,Z 494.217,A -85,B 0,C 180,E1 -4823.827,E2 -4823.827} C_VEL
LIN {X 0,Y 523.937,Z 494.218,A -85,B 0,C 180,E1 -4826.635,E2 -4826.635} C_VEL
LIN {X 0,Y 523.956,Z 494.217,A -85,B 0,C 180,E1 -4829.356,E2 -4829.356} C_VEL
LIN {X 0,Y 523.972,Z 494.212,A -85,B 0,C 180,E1 -4832.28,E2 -4832.28} C_VEL
LIN {X 0,Y 523.946,Z 494.215,A -85,B 0,C 180,E1 -4834.581,E2 -4834.581} C_VEL
LIN {X 0,Y 523.908,Z 494.222,A -85,B 0,C 180,E1 -4837.106,E2 -4837.106} C_VEL
LIN {X 0,Y 523.97,Z 494.212,A -85,B 0,C 180,E1 -4839.865,E2 -4839.865} C_VEL
LIN {X 0,Y 523.961,Z 494.214,A -85,B 0,C 180,E1 -4842.837,E2 -4842.837} C_VEL
LIN {X 0,Y 523.966,Z 494.219,A -85,B 0,C 180,E1 -4845.235,E2 -4845.235} C_VEL
LIN {X 0,Y 524.003,Z 494.208,A -85,B 0,C 180,E1 -4848.394,E2 -4848.394} C_VEL
LIN {X 0,Y 523.998,Z 494.205,A -85,B 0,C 180,E1 -4851.516,E2 -4851.516} C_VEL
LIN {X 0,Y 524.094,Z 494.198,A -85,B 0,C 180,E1 -4854.614,E2 -4854.614} C_VEL
LIN {X 0,Y 524.103,Z 494.195,A -85,B 0,C 180,E1 -4857.695,E2 -4857.695} C_VEL
LIN {X 0,Y 524.117,Z 494.189,A -85,B 0,C 180,E1 -4860.768,E2 -4860.768} C_VEL
LIN {X 0,Y 524.069,Z 494.207,A -85,B 0,C 180,E1 -4863.075,E2 -4863.075} C_VEL
LIN {X 0,Y 524.044,Z 494.201,A -85,B 0,C 180,E1 -4866.159,E2 -4866.159} C_VEL
LIN {X 0,Y 523.996,Z 494.213,A -85,B 0,C 180,E1 -4869.262,E2 -4869.262} C_VEL
LIN {X 0,Y 523.999,Z 494.209,A -85,B 0,C 180,E1 -4871.743,E2 -4871.743} C_VEL
LIN {X 0,Y 523.983,Z 494.214,A -85,B 0,C 180,E1 -4875.053,E2 -4875.053} C_VEL
LIN {X 0,Y 523.957,Z 494.212,A -85,B 0,C 180,E1 -4877.97,E2 -4877.97} C_VEL
LIN {X 0,Y 523.964,Z 494.214,A -85,B 0,C 180,E1 -4880.411,E2 -4880.411} C_VEL
LIN {X 0,Y 523.909,Z 494.224,A -85,B 0,C 180,E1 -4882.894,E2 -4882.894} C_VEL
LIN {X 0,Y 523.948,Z 494.219,A -85,B 0,C 180,E1 -4885.419,E2 -4885.419} C_VEL
LIN {X 0,Y 523.964,Z 494.212,A -85,B 0,C 180,E1 -4888,E2 -4888} C_VEL
LIN {X 0,Y 523.947,Z 494.218,A -85,B 0,C 180,E1 -4890.857,E2 -4890.857} C_VEL
LIN {X 0,Y 523.958,Z 494.213,A -85,B 0,C 180,E1 -4893.736,E2 -4893.736} C_VEL
LIN {X 0,Y 523.921,Z 494.219,A -85,B 0,C 180,E1 -4896.406,E2 -4896.406} C_VEL
LIN {X 0,Y 523.92,Z 494.225,A -85,B 0,C 180,E1 -4899.085,E2 -4899.085} C_VEL
LIN {X 0,Y 523.954,Z 494.216,A -85,B 0,C 180,E1 -4902.119,E2 -4902.119} C_VEL
LIN {X 0,Y 523.954,Z 494.22,A -85,B 0,C 180,E1 -4905.31,E2 -4905.31} C_VEL
LIN {X 0,Y 523.922,Z 494.224,A -85,B 0,C 180,E1 -4906.925,E2 -4906.925} C_VEL
LIN {X 0,Y 523.255,Z 494.305,A -85,B 0,C 180,E1 -4907.567,E2 -4907.567} C_VEL
LIN {X 0,Y 520.409,Z 494.66,A -85,B 0,C 180,E1 -4908.608,E2 -4908.608} C_VEL
LIN {X 0,Y 518.002,Z 494.958,A -85,B 0,C 180,E1 -4909.447,E2 -4909.447} C_VEL
LIN {X 0,Y 516.967,Z 495.085,A -85,B 0,C 180,E1 -4910.095,E2 -4910.095} C_VEL
LIN {X 0,Y 516.881,Z 495.096,A -85,B 0,C 180,E1 -4910.314,E2 -4910.314} C_VEL
LIN {X 0,Y 516.876,Z 495.1,A -85,B 0,C 180,E1 -4913.344,E2 -4913.344} C_VEL
LIN {X 0,Y 516.908,Z 495.093,A -85,B 0,C 180,E1 -4916.122,E2 -4916.122} C_VEL
LIN {X 0,Y 516.892,Z 495.101,A -85,B 0,C 180,E1 -4918.937,E2 -4918.937} C_VEL
LIN {X 0,Y 516.921,Z 495.093,A -85,B 0,C 180,E1 -4921.586,E2 -4921.586} C_VEL
LIN {X 0,Y 516.982,Z 495.234,A -85,B 0,C 180,E1 -4924.376,E2 -4924.376} C_VEL
LIN {X 0,Y 518.237,Z 502.941,A -85,B 0,C 180,E1 -4925.685,E2 -4925.685} C_VEL
LIN {X 0,Y 517.924,Z 519.149,A -85,B 0,C 180,E1 -4928.299,E2 -4928.299} C_VEL
LIN {X 0,Y 517.579,Z 537.097,A -85,B 0,C 180,E1 -4931.187,E2 -4931.187} C_VEL
LIN {X 0,Y 517.407,Z 546.614,A -85,B 0,C 180,E1 -4932.69,E2 -4932.69} C_VEL
LIN {X 0,Y 519.115,Z 557.018,A -85,B 0,C 180,E1 -4932.888,E2 -4932.888} C_VEL
LIN {X 0,Y 518.617,Z 654.122,A -85,B 0,C 180,E1 -4934.252,E2 -4934.252} C_VEL
LIN {X 0,Y 518.473,Z 667.343,A -85,B 0,C 180,E1 -4934.588,E2 -4934.588} C_VEL
LIN {X 0,Y 518.224,Z 679.813,A -85,B 0,C 180,E1 -4935.068,E2 -4935.068} C_VEL
LIN {X 0,Y 517.937,Z 691.256,A -85,B 0,C 180,E1 -4935.663,E2 -4935.663} C_VEL
LIN {X 0,Y 517.593,Z 703.112,A -85,B 0,C 180,E1 -4936.454,E2 -4936.454} C_VEL
LIN {X 0,Y 517.267,Z 713.589,A -85,B 0,C 180,E1 -4937.345,E2 -4937.345} C_VEL
LIN {X 0,Y 516.95,Z 723.923,A -85,B 0,C 180,E1 -4938.435,E2 -4938.435} C_VEL
LIN {X 0,Y 516.755,Z 732.818,A -85,B 0,C 180,E1 -4939.619,E2 -4939.619} C_VEL
LIN {X 0,Y 516.553,Z 739.988,A -85,B 0,C 180,E1 -4940.801,E2 -4940.801} C_VEL
LIN {X 0,Y 516.414,Z 746.553,A -85,B 0,C 180,E1 -4942.178,E2 -4942.178} C_VEL
LIN {X 0,Y 516.353,Z 751.345,A -85,B 0,C 180,E1 -4943.515,E2 -4943.515} C_VEL
LIN {X 0,Y 516.318,Z 754.094,A -85,B 0,C 180,E1 -4944.533,E2 -4944.533} C_VEL
LIN {X 0,Y 516.291,Z 756.904,A -85,B 0,C 180,E1 -4946.097,E2 -4946.097} C_VEL
LIN {X 0,Y 516.273,Z 757.698,A -85,B 0,C 180,E1 -4946.879,E2 -4946.879} C_VEL
LIN {X 0,Y 516.26,Z 758.073,A -85,B 0,C 180,E1 -4947.659,E2 -4947.659} C_VEL
LIN {X 0,Y 516.16,Z 757.696,A -85,B 0,C 180,E1 -4949.22,E2 -4949.22} C_VEL
LIN {X 0,Y 516.157,Z 756.898,A -85,B 0,C 180,E1 -4950,E2 -4950} C_VEL
LIN {X 0,Y 516.222,Z 754.093,A -85,B 0,C 180,E1 -4951.56,E2 -4951.56} C_VEL
LIN {X 0,Y 516.348,Z 750.867,A -85,B 0,C 180,E1 -4952.73,E2 -4952.73} C_VEL
LIN {X 0,Y 516.428,Z 746.592,A -85,B 0,C 180,E1 -4953.902,E2 -4953.902} C_VEL
LIN {X 0,Y 516.586,Z 740.099,A -85,B 0,C 180,E1 -4955.269,E2 -4955.269} C_VEL
LIN {X 0,Y 516.792,Z 732.859,A -85,B 0,C 180,E1 -4956.465,E2 -4956.465} C_VEL
LIN {X 0,Y 516.97,Z 724.235,A -85,B 0,C 180,E1 -4957.617,E2 -4957.617} C_VEL
LIN {X 0,Y 517.276,Z 714.113,A -85,B 0,C 180,E1 -4958.693,E2 -4958.693} C_VEL
LIN {X 0,Y 517.61,Z 703.88,A -85,B 0,C 180,E1 -4959.574,E2 -4959.574} C_VEL
LIN {X 0,Y 517.88,Z 694.051,A -85,B 0,C 180,E1 -4960.26,E2 -4960.26} C_VEL
LIN {X 0,Y 518.154,Z 682.49,A -85,B 0,C 180,E1 -4960.897,E2 -4960.897} C_VEL
LIN {X 0,Y 518.431,Z 669.335,A -85,B 0,C 180,E1 -4961.435,E2 -4961.435} C_VEL
LIN {X 0,Y 518.594,Z 657.137,A -85,B 0,C 180,E1 -4961.778,E2 -4961.778} C_VEL
LIN {X 0,Y 518.76,Z 638.423,A -85,B 0,C 180,E1 -4962.072,E2 -4962.072} C_VEL
LIN {X 0,Y 519.033,Z 556.15,A -85,B 0,C 180,E1 -4963.217,E2 -4963.217} C_VEL
LIN {X 0,Y 517.364,Z 546.269,A -85,B 0,C 180,E1 -4963.427,E2 -4963.427} C_VEL
LIN {X 0,Y 517.735,Z 529.329,A -85,B 0,C 180,E1 -4966.157,E2 -4966.157} C_VEL
LIN {X 0,Y 518.113,Z 510.415,A -85,B 0,C 180,E1 -4969.204,E2 -4969.204} C_VEL
LIN {X 0,Y 518.137,Z 501.517,A -85,B 0,C 180,E1 -4970.65,E2 -4970.65} C_VEL
LIN {X 0,Y 516.915,Z 495.098,A -85,B 0,C 180,E1 -4971.745,E2 -4971.745} C_VEL
LIN {X 0,Y 516.911,Z 495.103,A -85,B 0,C 180,E1 -4974.927,E2 -4974.927} C_VEL
LIN {X 0,Y 516.927,Z 495.091,A -85,B 0,C 180,E1 -4977.904,E2 -4977.904} C_VEL
LIN {X 0,Y 516.895,Z 495.096,A -85,B 0,C 180,E1 -4980.203,E2 -4980.203} C_VEL
LIN {X 0,Y 516.898,Z 495.102,A -85,B 0,C 180,E1 -4982.946,E2 -4982.946} C_VEL
LIN {X 0,Y 516.872,Z 495.097,A -85,B 0,C 180,E1 -4985.779,E2 -4985.779} C_VEL
LIN {X 0,Y 516.883,Z 495.101,A -85,B 0,C 180,E1 -4988.715,E2 -4988.715} C_VEL
LIN {X 0,Y 516.915,Z 495.091,A -85,B 0,C 180,E1 -4991.774,E2 -4991.774} C_VEL
LIN {X 0,Y 516.92,Z 495.093,A -85,B 0,C 180,E1 -4995.009,E2 -4995.009} C_VEL
LIN {X 0,Y 516.914,Z 495.094,A -85,B 0,C 180,E1 -4998.397,E2 -4998.397} C_VEL
LIN {X 0,Y 516.879,Z 495.099,A -85,B 0,C 180,E1 -5001.283,E2 -5001.283} C_VEL
LIN {X 0,Y 516.886,Z 495.098,A -85,B 0,C 180,E1 -5004.22,E2 -5004.22} C_VEL
LIN {X 0,Y 516.963,Z 495.091,A -85,B 0,C 180,E1 -5007.564,E2 -5007.564} C_VEL
LIN {X 0,Y 517.129,Z 498.784,A -85,B 0,C 180,E1 -5008.45,E2 -5008.45} C_VEL
LIN {X 0,Y 517.124,Z 499.838,A -85,B 0,C 180,E1 -5008.695,E2 -5008.695} C_VEL
LIN {X 0,Y 519.139,Z 510.208,A -85,B 0,C 180,E1 -5008.917,E2 -5008.917} C_VEL
LIN {X 0,Y 518.599,Z 605.774,A -85,B 0,C 180,E1 -5010.301,E2 -5010.301} C_VEL
LIN {X 0,Y 518.437,Z 618.291,A -85,B 0,C 180,E1 -5010.623,E2 -5010.623} C_VEL
LIN {X 0,Y 518.172,Z 632.026,A -85,B 0,C 180,E1 -5011.162,E2 -5011.162} C_VEL
LIN {X 0,Y 517.894,Z 643.43,A -85,B 0,C 180,E1 -5011.775,E2 -5011.775} C_VEL
LIN {X 0,Y 517.563,Z 654.143,A -85,B 0,C 180,E1 -5012.504,E2 -5012.504} C_VEL
LIN {X 0,Y 517.321,Z 664.301,A -85,B 0,C 180,E1 -5013.364,E2 -5013.364} C_VEL
LIN {X 0,Y 517.013,Z 674.437,A -85,B 0,C 180,E1 -5014.431,E2 -5014.431} C_VEL
LIN {X 0,Y 516.797,Z 682.036,A -85,B 0,C 180,E1 -5015.418,E2 -5015.418} C_VEL
LIN {X 0,Y 516.586,Z 689.172,A -85,B 0,C 180,E1 -5016.55,E2 -5016.55} C_VEL
LIN {X 0,Y 516.481,Z 695.068,A -85,B 0,C 180,E1 -5017.711,E2 -5017.711} C_VEL
LIN {X 0,Y 516.365,Z 699.725,A -85,B 0,C 180,E1 -5018.858,E2 -5018.858} C_VEL
LIN {X 0,Y 516.301,Z 703.605,A -85,B 0,C 180,E1 -5020.104,E2 -5020.104} C_VEL
LIN {X 0,Y 516.207,Z 705.517,A -85,B 0,C 180,E1 -5020.928,E2 -5020.928} C_VEL
LIN {X 0,Y 516.194,Z 707.014,A -85,B 0,C 180,E1 -5021.751,E2 -5021.751} C_VEL
LIN {X 0,Y 516.215,Z 708.016,A -85,B 0,C 180,E1 -5022.571,E2 -5022.571} C_VEL
LIN {X 0,Y 516.171,Z 708.697,A -85,B 0,C 180,E1 -5024.198,E2 -5024.198} C_VEL
LIN {X 0,Y 516.222,Z 708.353,A -85,B 0,C 180,E1 -5025.148,E2 -5025.148} C_VEL
LIN {X 0,Y 516.208,Z 706.569,A -85,B 0,C 180,E1 -5026.617,E2 -5026.617} C_VEL
LIN {X 0,Y 516.313,Z 704.063,A -85,B 0,C 180,E1 -5027.82,E2 -5027.82} C_VEL
LIN {X 0,Y 516.371,Z 700.551,A -85,B 0,C 180,E1 -5029.015,E2 -5029.015} C_VEL
LIN {X 0,Y 516.471,Z 695.941,A -85,B 0,C 180,E1 -5030.206,E2 -5030.206} C_VEL
LIN {X 0,Y 516.661,Z 689.018,A -85,B 0,C 180,E1 -5031.591,E2 -5031.591} C_VEL
LIN {X 0,Y 516.854,Z 681.447,A -85,B 0,C 180,E1 -5032.774,E2 -5032.774} C_VEL
LIN {X 0,Y 517.059,Z 673.706,A -85,B 0,C 180,E1 -5033.757,E2 -5033.757} C_VEL
LIN {X 0,Y 517.275,Z 664.312,A -85,B 0,C 180,E1 -5034.738,E2 -5034.738} C_VEL
LIN {X 0,Y 517.582,Z 653.891,A -85,B 0,C 180,E1 -5035.619,E2 -5035.619} C_VEL
LIN {X 0,Y 517.902,Z 642.241,A -85,B 0,C 180,E1 -5036.401,E2 -5036.401} C_VEL
LIN {X 0,Y 518.211,Z 629.736,A -85,B 0,C 180,E1 -5037.036,E2 -5037.036} C_VEL
LIN {X 0,Y 518.415,Z 617.275,A -85,B 0,C 180,E1 -5037.499,E2 -5037.499} C_VEL
LIN {X 0,Y 518.593,Z 604.426,A -85,B 0,C 180,E1 -5037.815,E2 -5037.815} C_VEL
LIN {X 0,Y 519.065,Z 509.894,A -85,B 0,C 180,E1 -5039.176,E2 -5039.176} C_VEL
LIN {X 0,Y 517.201,Z 500.676,A -85,B 0,C 180,E1 -5039.367,E2 -5039.367} C_VEL
LIN {X 0,Y 517.09,Z 495.077,A -85,B 0,C 180,E1 -5040.73,E2 -5040.73} C_VEL
LIN {X 0,Y 517.009,Z 495.087,A -85,B 0,C 180,E1 -5043.117,E2 -5043.117} C_VEL
LIN {X 0,Y 517.006,Z 495.082,A -85,B 0,C 180,E1 -5046.243,E2 -5046.243} C_VEL
LIN {X 0,Y 516.95,Z 495.095,A -85,B 0,C 180,E1 -5049.389,E2 -5049.389} C_VEL
LIN {X 0,Y 516.973,Z 495.087,A -85,B 0,C 180,E1 -5051.824,E2 -5051.824} C_VEL
LIN {X 0,Y 516.934,Z 495.097,A -85,B 0,C 180,E1 -5055.147,E2 -5055.147} C_VEL
LIN {X 0,Y 516.917,Z 495.091,A -85,B 0,C 180,E1 -5058.222,E2 -5058.222} C_VEL
LIN {X 0,Y 516.904,Z 495.095,A -85,B 0,C 180,E1 -5060.702,E2 -5060.702} C_VEL
LIN {X 0,Y 516.902,Z 495.093,A -85,B 0,C 180,E1 -5064.072,E2 -5064.072} C_VEL
LIN {X 0,Y 516.921,Z 495.092,A -85,B 0,C 180,E1 -5066.658,E2 -5066.658} C_VEL
LIN {X 0,Y 516.917,Z 495.092,A -85,B 0,C 180,E1 -5069.527,E2 -5069.527} C_VEL
LIN {X 0,Y 516.894,Z 495.094,A -85,B 0,C 180,E1 -5072.545,E2 -5072.545} C_VEL
LIN {X 0,Y 516.877,Z 495.099,A -85,B 0,C 180,E1 -5075.333,E2 -5075.333} C_VEL
LIN {X 0,Y 516.876,Z 495.095,A -85,B 0,C 180,E1 -5077.944,E2 -5077.944} C_VEL
LIN {X 0,Y 516.88,Z 495.1,A -85,B 0,C 180,E1 -5080.742,E2 -5080.742} C_VEL
LIN {X 0,Y 516.879,Z 495.102,A -85,B 0,C 180,E1 -5082.832,E2 -5082.832} C_VEL
LIN {X 0,Y 516.918,Z 495.099,A -85,B 0,C 180,E1 -5085.011,E2 -5085.011} C_VEL
LIN {X 0,Y 516.914,Z 495.095,A -85,B 0,C 180,E1 -5088.399,E2 -5088.399} C_VEL
LIN {X 0,Y 516.88,Z 495.1,A -85,B 0,C 180,E1 -5091.285,E2 -5091.285} C_VEL
LIN {X 0,Y 516.885,Z 495.097,A -85,B 0,C 180,E1 -5094.222,E2 -5094.222} C_VEL
LIN {X 0,Y 516.896,Z 495.103,A -85,B 0,C 180,E1 -5097.054,E2 -5097.054} C_VEL
LIN {X 0,Y 516.892,Z 495.098,A -85,B 0,C 180,E1 -5099.797,E2 -5099.797} C_VEL
LIN {X 0,Y 516.928,Z 495.097,A -85,B 0,C 180,E1 -5102.468,E2 -5102.468} C_VEL
LIN {X 0,Y 516.967,Z 495.267,A -85,B 0,C 180,E1 -5103.649,E2 -5103.649} C_VEL
LIN {X 0,Y 518.915,Z 506.033,A -85,B 0,C 180,E1 -5105.288,E2 -5105.288} C_VEL
LIN {X 0,Y 518.394,Z 526.017,A -85,B 0,C 180,E1 -5108.111,E2 -5108.111} C_VEL
LIN {X 0,Y 517.926,Z 546.764,A -85,B 0,C 180,E1 -5110.994,E2 -5110.994} C_VEL
LIN {X 0,Y 517.45,Z 570.44,A -85,B 0,C 180,E1 -5114.239,E2 -5114.239} C_VEL
LIN {X 0,Y 517.409,Z 573.279,A -85,B 0,C 180,E1 -5114.627,E2 -5114.627} C_VEL
LIN {X 0,Y 519.032,Z 585.557,A -85,B 0,C 180,E1 -5114.867,E2 -5114.867} C_VEL
LIN {X 0,Y 518.585,Z 682.228,A -85,B 0,C 180,E1 -5116.231,E2 -5116.231} C_VEL
LIN {X 0,Y 518.309,Z 695.713,A -85,B 0,C 180,E1 -5116.573,E2 -5116.573} C_VEL
LIN {X 0,Y 518.066,Z 708.612,A -85,B 0,C 180,E1 -5117.066,E2 -5117.066} C_VEL
LIN {X 0,Y 517.795,Z 720.883,A -85,B 0,C 180,E1 -5117.706,E2 -5117.706} C_VEL
LIN {X 0,Y 517.509,Z 731.906,A -85,B 0,C 180,E1 -5118.445,E2 -5118.445} C_VEL
LIN {X 0,Y 517.199,Z 742.54,A -85,B 0,C 180,E1 -5119.331,E2 -5119.331} C_VEL
LIN {X 0,Y 516.968,Z 751.222,A -85,B 0,C 180,E1 -5120.216,E2 -5120.216} C_VEL
LIN {X 0,Y 516.759,Z 759.234,A -85,B 0,C 180,E1 -5121.199,E2 -5121.199} C_VEL
LIN {X 0,Y 516.562,Z 767.063,A -85,B 0,C 180,E1 -5122.377,E2 -5122.377} C_VEL
LIN {X 0,Y 516.421,Z 772.826,A -85,B 0,C 180,E1 -5123.445,E2 -5123.445} C_VEL
LIN {X 0,Y 516.405,Z 777.602,A -85,B 0,C 180,E1 -5124.533,E2 -5124.533} C_VEL
LIN {X 0,Y 516.326,Z 781.624,A -85,B 0,C 180,E1 -5125.707,E2 -5125.707} C_VEL
LIN {X 0,Y 516.282,Z 784.595,A -85,B 0,C 180,E1 -5126.879,E2 -5126.879} C_VEL
LIN {X 0,Y 516.26,Z 786.01,A -85,B 0,C 180,E1 -5127.659,E2 -5127.659} C_VEL
LIN {X 0,Y 516.16,Z 787.625,A -85,B 0,C 180,E1 -5129.22,E2 -5129.22} C_VEL
LIN {X 0,Y 516.154,Z 787.843,A -85,B 0,C 180,E1 -5130,E2 -5130} C_VEL
LIN {X 0,Y 516.191,Z 787.013,A -85,B 0,C 180,E1 -5131.56,E2 -5131.56} C_VEL
LIN {X 0,Y 516.26,Z 786.011,A -85,B 0,C 180,E1 -5132.341,E2 -5132.341} C_VEL
LIN {X 0,Y 516.282,Z 784.599,A -85,B 0,C 180,E1 -5133.121,E2 -5133.121} C_VEL
LIN {X 0,Y 516.326,Z 781.636,A -85,B 0,C 180,E1 -5134.293,E2 -5134.293} C_VEL
LIN {X 0,Y 516.405,Z 777.622,A -85,B 0,C 180,E1 -5135.467,E2 -5135.467} C_VEL
LIN {X 0,Y 516.444,Z 772.264,A -85,B 0,C 180,E1 -5136.679,E2 -5136.679} C_VEL
LIN {X 0,Y 516.578,Z 765.932,A -85,B 0,C 180,E1 -5137.819,E2 -5137.819} C_VEL
LIN {X 0,Y 516.787,Z 757.813,A -85,B 0,C 180,E1 -5138.997,E2 -5138.997} C_VEL
LIN {X 0,Y 517.019,Z 749.535,A -85,B 0,C 180,E1 -5139.98,E2 -5139.98} C_VEL
LIN {X 0,Y 517.298,Z 739.417,A -85,B 0,C 180,E1 -5140.964,E2 -5140.964} C_VEL
LIN {X 0,Y 517.571,Z 729.443,A -85,B 0,C 180,E1 -5141.752,E2 -5141.752} C_VEL
LIN {X 0,Y 517.883,Z 718.048,A -85,B 0,C 180,E1 -5142.471,E2 -5142.471} C_VEL
LIN {X 0,Y 518.158,Z 705.542,A -85,B 0,C 180,E1 -5143.081,E2 -5143.081} C_VEL
LIN {X 0,Y 518.387,Z 692.997,A -85,B 0,C 180,E1 -5143.524,E2 -5143.524} C_VEL
LIN {X 0,Y 518.597,Z 679.93,A -85,B 0,C 180,E1 -5143.819,E2 -5143.819} C_VEL
LIN {X 0,Y 519.003,Z 584.925,A -85,B 0,C 180,E1 -5145.153,E2 -5145.153} C_VEL
LIN {X 0,Y 517.461,Z 573.809,A -85,B 0,C 180,E1 -5145.372,E2 -5145.372} C_VEL
LIN {X 0,Y 517.934,Z 550.891,A -85,B 0,C 180,E1 -5148.554,E2 -5148.554} C_VEL
LIN {X 0,Y 518.539,Z 528.562,A -85,B 0,C 180,E1 -5151.674,E2 -5151.674} C_VEL
LIN {X 0,Y 519.088,Z 507.996,A -85,B 0,C 180,E1 -5154.602,E2 -5154.602} C_VEL
LIN {X 0,Y 518.686,Z 503.596,A -85,B 0,C 180,E1 -5155.264,E2 -5155.264} C_VEL
LIN {X 0,Y 516.941,Z 495.094,A -85,B 0,C 180,E1 -5156.626,E2 -5156.626} C_VEL
LIN {X 0,Y 516.91,Z 495.098,A -85,B 0,C 180,E1 -5159.523,E2 -5159.523} C_VEL
LIN {X 0,Y 516.897,Z 495.096,A -85,B 0,C 180,E1 -5162.543,E2 -5162.543} C_VEL
LIN {X 0,Y 516.865,Z 495.103,A -85,B 0,C 180,E1 -5165.329,E2 -5165.329} C_VEL
LIN {X 0,Y 516.878,Z 495.085,A -85,B 0,C 180,E1 -5167.942,E2 -5167.942} C_VEL
LIN {X 0,Y 516.882,Z 495.096,A -85,B 0,C 180,E1 -5170.741,E2 -5170.741} C_VEL
LIN {X 0,Y 516.901,Z 495.097,A -85,B 0,C 180,E1 -5172.828,E2 -5172.828} C_VEL
LIN {X 0,Y 516.918,Z 495.096,A -85,B 0,C 180,E1 -5175.009,E2 -5175.009} C_VEL
LIN {X 0,Y 516.917,Z 495.088,A -85,B 0,C 180,E1 -5178.397,E2 -5178.397} C_VEL
LIN {X 0,Y 516.877,Z 495.102,A -85,B 0,C 180,E1 -5181.284,E2 -5181.284} C_VEL
LIN {X 0,Y 516.884,Z 495.092,A -85,B 0,C 180,E1 -5184.221,E2 -5184.221} C_VEL
LIN {X 0,Y 516.891,Z 495.102,A -85,B 0,C 180,E1 -5187.053,E2 -5187.053} C_VEL
LIN {X 0,Y 516.894,Z 495.091,A -85,B 0,C 180,E1 -5189.796,E2 -5189.796} C_VEL
LIN {X 0,Y 516.922,Z 495.091,A -85,B 0,C 180,E1 -5192.467,E2 -5192.467} C_VEL
LIN {X 0,Y 516.903,Z 495.095,A -85,B 0,C 180,E1 -5195.072,E2 -5195.072} C_VEL
LIN {X 0,Y 516.877,Z 495.095,A -85,B 0,C 180,E1 -5198.462,E2 -5198.462} C_VEL
LIN {X 0,Y 516.897,Z 495.099,A -85,B 0,C 180,E1 -5200.955,E2 -5200.955} C_VEL
LIN {X 0,Y 516.908,Z 495.09,A -85,B 0,C 180,E1 -5203.41,E2 -5203.41} C_VEL
LIN {X 0,Y 516.885,Z 495.094,A -85,B 0,C 180,E1 -5205.833,E2 -5205.833} C_VEL
LIN {X 0,Y 516.994,Z 495.081,A -85,B 0,C 180,E1 -5208.234,E2 -5208.234} C_VEL
LIN {X 0,Y 516.963,Z 495.082,A -85,B 0,C 180,E1 -5211.4,E2 -5211.4} C_VEL
LIN {X 0,Y 517.054,Z 495.074,A -85,B 0,C 180,E1 -5214.54,E2 -5214.54} C_VEL
LIN {X 0,Y 517.075,Z 495.07,A -85,B 0,C 180,E1 -5217.663,E2 -5217.663} C_VEL
LIN {X 0,Y 517.087,Z 495.064,A -85,B 0,C 180,E1 -5220.779,E2 -5220.779} C_VEL
LIN {X 0,Y 517.01,Z 495.087,A -85,B 0,C 180,E1 -5223.117,E2 -5223.117} C_VEL
LIN {X 0,Y 517.006,Z 495.078,A -85,B 0,C 180,E1 -5226.243,E2 -5226.243} C_VEL
LIN {X 0,Y 516.95,Z 495.088,A -85,B 0,C 180,E1 -5229.39,E2 -5229.39} C_VEL
LIN {X 0,Y 516.948,Z 495.087,A -85,B 0,C 180,E1 -5231.811,E2 -5231.811} C_VEL
LIN {X 0,Y 516.935,Z 495.089,A -85,B 0,C 180,E1 -5235.147,E2 -5235.147} C_VEL
LIN {X 0,Y 516.919,Z 495.089,A -85,B 0,C 180,E1 -5238.223,E2 -5238.223} C_VEL
LIN {X 0,Y 516.905,Z 495.096,A -85,B 0,C 180,E1 -5240.702,E2 -5240.702} C_VEL
LIN {X 0,Y 516.904,Z 495.088,A -85,B 0,C 180,E1 -5244.073,E2 -5244.073} C_VEL
LIN {X 0,Y 516.923,Z 495.094,A -85,B 0,C 180,E1 -5246.658,E2 -5246.658} C_VEL
LIN {X 0,Y 516.918,Z 495.089,A -85,B 0,C 180,E1 -5249.527,E2 -5249.527} C_VEL
LIN {X 0,Y 516.895,Z 495.096,A -85,B 0,C 180,E1 -5252.545,E2 -5252.545} C_VEL
LIN {X 0,Y 516.879,Z 495.1,A -85,B 0,C 180,E1 -5255.334,E2 -5255.334} C_VEL
LIN {X 0,Y 516.881,Z 495.096,A -85,B 0,C 180,E1 -5257.945,E2 -5257.945} C_VEL
LIN {X 0,Y 516.882,Z 495.099,A -85,B 0,C 180,E1 -5260.742,E2 -5260.742} C_VEL
LIN {X 0,Y 516.9,Z 495.101,A -85,B 0,C 180,E1 -5262.83,E2 -5262.83} C_VEL
LIN {X 0,Y 516.92,Z 495.1,A -85,B 0,C 180,E1 -5265.011,E2 -5265.011} C_VEL
LIN {X 0,Y 516.916,Z 495.093,A -85,B 0,C 180,E1 -5268.399,E2 -5268.399} C_VEL
LIN {X 0,Y 516.881,Z 495.096,A -85,B 0,C 180,E1 -5270.314,E2 -5270.314} C_VEL
LIN {X 0,Y 516.213,Z 495.187,A -85,B 0,C 180,E1 -5270.965,E2 -5270.965} C_VEL
LIN {X 0,Y 513.364,Z 495.54,A -85,B 0,C 180,E1 -5272.02,E2 -5272.02} C_VEL
LIN {X 0,Y 510.953,Z 495.841,A -85,B 0,C 180,E1 -5272.871,E2 -5272.871} C_VEL
LIN {X 0,Y 509.909,Z 495.966,A -85,B 0,C 180,E1 -5273.527,E2 -5273.527} C_VEL
LIN {X 0,Y 509.819,Z 495.976,A -85,B 0,C 180,E1 -5273.75,E2 -5273.75} C_VEL
LIN {X 0,Y 509.859,Z 495.973,A -85,B 0,C 180,E1 -5276.54,E2 -5276.54} C_VEL
LIN {X 0,Y 509.847,Z 495.977,A -85,B 0,C 180,E1 -5279.335,E2 -5279.335} C_VEL
LIN {X 0,Y 509.894,Z 495.967,A -85,B 0,C 180,E1 -5282.055,E2 -5282.055} C_VEL
LIN {X 0,Y 509.938,Z 496.114,A -85,B 0,C 180,E1 -5284.216,E2 -5284.216} C_VEL
LIN {X 0,Y 511.309,Z 504.468,A -85,B 0,C 180,E1 -5285.648,E2 -5285.648} C_VEL
LIN {X 0,Y 510.94,Z 522.682,A -85,B 0,C 180,E1 -5288.623,E2 -5288.623} C_VEL
LIN {X 0,Y 510.484,Z 544.103,A -85,B 0,C 180,E1 -5292.075,E2 -5292.075} C_VEL
LIN {X 0,Y 510.431,Z 546.622,A -85,B 0,C 180,E1 -5292.471,E2 -5292.471} C_VEL
LIN {X 0,Y 512.279,Z 557.806,A -85,B 0,C 180,E1 -5292.691,E2 -5292.691} C_VEL
LIN {X 0,Y 511.736,Z 654.841,A -85,B 0,C 180,E1 -5294.076,E2 -5294.076} C_VEL
LIN {X 0,Y 511.578,Z 667.571,A -85,B 0,C 180,E1 -5294.406,E2 -5294.406} C_VEL
LIN {X 0,Y 511.308,Z 680.446,A -85,B 0,C 180,E1 -5294.913,E2 -5294.913} C_VEL
LIN {X 0,Y 510.968,Z 692.642,A -85,B 0,C 180,E1 -5295.564,E2 -5295.564} C_VEL
LIN {X 0,Y 510.614,Z 702.917,A -85,B 0,C 180,E1 -5296.266,E2 -5296.266} C_VEL
LIN {X 0,Y 510.294,Z 713.483,A -85,B 0,C 180,E1 -5297.169,E2 -5297.169} C_VEL
LIN {X 0,Y 509.961,Z 723.668,A -85,B 0,C 180,E1 -5298.251,E2 -5298.251} C_VEL
LIN {X 0,Y 509.783,Z 731.486,A -85,B 0,C 180,E1 -5299.274,E2 -5299.274} C_VEL
LIN {X 0,Y 509.507,Z 738.937,A -85,B 0,C 180,E1 -5300.473,E2 -5300.473} C_VEL
LIN {X 0,Y 509.38,Z 744.914,A -85,B 0,C 180,E1 -5301.67,E2 -5301.67} C_VEL
LIN {X 0,Y 509.317,Z 749.635,A -85,B 0,C 180,E1 -5302.866,E2 -5302.866} C_VEL
LIN {X 0,Y 509.231,Z 753.241,A -85,B 0,C 180,E1 -5304.059,E2 -5304.059} C_VEL
LIN {X 0,Y 509.142,Z 755.84,A -85,B 0,C 180,E1 -5305.249,E2 -5305.249} C_VEL
LIN {X 0,Y 509.187,Z 757.057,A -85,B 0,C 180,E1 -5306.043,E2 -5306.043} C_VEL
LIN {X 0,Y 509.189,Z 757.872,A -85,B 0,C 180,E1 -5306.835,E2 -5306.835} C_VEL
LIN {X 0,Y 509.189,Z 758.258,A -85,B 0,C 180,E1 -5307.627,E2 -5307.627} C_VEL
LIN {X 0,Y 509.074,Z 757.903,A -85,B 0,C 180,E1 -5309.209,E2 -5309.209} C_VEL
LIN {X 0,Y 509.068,Z 757.126,A -85,B 0,C 180,E1 -5310,E2 -5310} C_VEL
LIN {X 0,Y 509.143,Z 754.343,A -85,B 0,C 180,E1 -5311.582,E2 -5311.582} C_VEL
LIN {X 0,Y 509.278,Z 751.139,A -85,B 0,C 180,E1 -5312.768,E2 -5312.768} C_VEL
LIN {X 0,Y 509.361,Z 746.888,A -85,B 0,C 180,E1 -5313.956,E2 -5313.956} C_VEL
LIN {X 0,Y 509.554,Z 741.468,A -85,B 0,C 180,E1 -5315.143,E2 -5315.143} C_VEL
LIN {X 0,Y 509.697,Z 734.69,A -85,B 0,C 180,E1 -5316.333,E2 -5316.333} C_VEL
LIN {X 0,Y 509.92,Z 726.211,A -85,B 0,C 180,E1 -5317.523,E2 -5317.523} C_VEL
LIN {X 0,Y 510.184,Z 717.548,A -85,B 0,C 180,E1 -5318.516,E2 -5318.516} C_VEL
LIN {X 0,Y 510.53,Z 708.062,A -85,B 0,C 180,E1 -5319.408,E2 -5319.408} C_VEL
LIN {X 0,Y 510.811,Z 697.631,A -85,B 0,C 180,E1 -5320.203,E2 -5320.203} C_VEL
LIN {X 0,Y 511.187,Z 686.091,A -85,B 0,C 180,E1 -5320.897,E2 -5320.897} C_VEL
LIN {X 0,Y 511.441,Z 674.274,A -85,B 0,C 180,E1 -5321.443,E2 -5321.443} C_VEL
LIN {X 0,Y 511.657,Z 661.352,A -85,B 0,C 180,E1 -5321.865,E2 -5321.865} C_VEL
LIN {X 0,Y 511.822,Z 647.545,A -85,B 0,C 180,E1 -5322.137,E2 -5322.137} C_VEL
LIN {X 0,Y 512.137,Z 556.622,A -85,B 0,C 180,E1 -5323.42,E2 -5323.42} C_VEL
LIN {X 0,Y 510.383,Z 546.427,A -85,B 0,C 180,E1 -5323.639,E2 -5323.639} C_VEL
LIN {X 0,Y 510.757,Z 530.683,A -85,B 0,C 180,E1 -5326.179,E2 -5326.179} C_VEL
LIN {X 0,Y 511.166,Z 510.428,A -85,B 0,C 180,E1 -5329.476,E2 -5329.476} C_VEL
LIN {X 0,Y 511.258,Z 503.307,A -85,B 0,C 180,E1 -5330.639,E2 -5330.639} C_VEL
LIN {X 0,Y 509.882,Z 495.973,A -85,B 0,C 180,E1 -5331.921,E2 -5331.921} C_VEL
LIN {X 0,Y 509.879,Z 495.976,A -85,B 0,C 180,E1 -5335.295,E2 -5335.295} C_VEL
LIN {X 0,Y 509.899,Z 495.967,A -85,B 0,C 180,E1 -5338.1,E2 -5338.1} C_VEL
LIN {X 0,Y 509.849,Z 495.978,A -85,B 0,C 180,E1 -5341.279,E2 -5341.279} C_VEL
LIN {X 0,Y 509.858,Z 495.97,A -85,B 0,C 180,E1 -5344.202,E2 -5344.202} C_VEL
LIN {X 0,Y 509.816,Z 495.979,A -85,B 0,C 180,E1 -5347.34,E2 -5347.34} C_VEL
LIN {X 0,Y 509.838,Z 495.973,A -85,B 0,C 180,E1 -5350.381,E2 -5350.381} C_VEL
LIN {X 0,Y 509.838,Z 495.978,A -85,B 0,C 180,E1 -5353.063,E2 -5353.063} C_VEL
LIN {X 0,Y 509.828,Z 495.971,A -85,B 0,C 180,E1 -5355.791,E2 -5355.791} C_VEL
LIN {X 0,Y 509.855,Z 495.976,A -85,B 0,C 180,E1 -5358.574,E2 -5358.574} C_VEL
LIN {X 0,Y 509.849,Z 495.972,A -85,B 0,C 180,E1 -5361.785,E2 -5361.785} C_VEL
LIN {X 0,Y 509.842,Z 495.98,A -85,B 0,C 180,E1 -5364.622,E2 -5364.622} C_VEL
LIN {X 0,Y 509.917,Z 495.974,A -85,B 0,C 180,E1 -5367.484,E2 -5367.484} C_VEL
LIN {X 0,Y 510.166,Z 499.058,A -85,B 0,C 180,E1 -5368.201,E2 -5368.201} C_VEL
LIN {X 0,Y 510.183,Z 500.456,A -85,B 0,C 180,E1 -5368.497,E2 -5368.497} C_VEL
LIN {X 0,Y 512.262,Z 510.718,A -85,B 0,C 180,E1 -5368.713,E2 -5368.713} C_VEL
LIN {X 0,Y 511.676,Z 606.698,A -85,B 0,C 180,E1 -5370.131,E2 -5370.131} C_VEL
LIN {X 0,Y 511.443,Z 620.858,A -85,B 0,C 180,E1 -5370.52,E2 -5370.52} C_VEL
LIN {X 0,Y 511.251,Z 632.883,A -85,B 0,C 180,E1 -5371.015,E2 -5371.015} C_VEL
LIN {X 0,Y 510.988,Z 643.591,A -85,B 0,C 180,E1 -5371.598,E2 -5371.598} C_VEL
LIN {X 0,Y 510.65,Z 654.183,A -85,B 0,C 180,E1 -5372.322,E2 -5372.322} C_VEL
LIN {X 0,Y 510.369,Z 663.856,A -85,B 0,C 180,E1 -5373.141,E2 -5373.141} C_VEL
LIN {X 0,Y 510.097,Z 672.767,A -85,B 0,C 180,E1 -5374.059,E2 -5374.059} C_VEL
LIN {X 0,Y 509.829,Z 681.666,A -85,B 0,C 180,E1 -5375.181,E2 -5375.181} C_VEL
LIN {X 0,Y 509.581,Z 689.514,A -85,B 0,C 180,E1 -5376.424,E2 -5376.424} C_VEL
LIN {X 0,Y 509.449,Z 695.257,A -85,B 0,C 180,E1 -5377.557,E2 -5377.557} C_VEL
LIN {X 0,Y 509.312,Z 699.386,A -85,B 0,C 180,E1 -5378.551,E2 -5378.551} C_VEL
LIN {X 0,Y 509.251,Z 703.484,A -85,B 0,C 180,E1 -5379.817,E2 -5379.817} C_VEL
LIN {X 0,Y 509.159,Z 705.593,A -85,B 0,C 180,E1 -5380.653,E2 -5380.653} C_VEL
LIN {X 0,Y 509.118,Z 707.201,A -85,B 0,C 180,E1 -5381.488,E2 -5381.488} C_VEL
LIN {X 0,Y 509.143,Z 708.303,A -85,B 0,C 180,E1 -5382.321,E2 -5382.321} C_VEL
LIN {X 0,Y 509.102,Z 709.282,A -85,B 0,C 180,E1 -5383.973,E2 -5383.973} C_VEL
LIN {X 0,Y 509.129,Z 708.952,A -85,B 0,C 180,E1 -5385.073,E2 -5385.073} C_VEL
LIN {X 0,Y 509.135,Z 707.518,A -85,B 0,C 180,E1 -5386.428,E2 -5386.428} C_VEL
LIN {X 0,Y 509.2,Z 706.078,A -85,B 0,C 180,E1 -5387.242,E2 -5387.242} C_VEL
LIN {X 0,Y 509.287,Z 703.114,A -85,B 0,C 180,E1 -5388.451,E2 -5388.451} C_VEL
LIN {X 0,Y 509.372,Z 699.057,A -85,B 0,C 180,E1 -5389.667,E2 -5389.667} C_VEL
LIN {X 0,Y 509.498,Z 692.841,A -85,B 0,C 180,E1 -5391.072,E2 -5391.072} C_VEL
LIN {X 0,Y 509.734,Z 686.046,A -85,B 0,C 180,E1 -5392.274,E2 -5392.274} C_VEL
LIN {X 0,Y 509.957,Z 677.887,A -85,B 0,C 180,E1 -5393.441,E2 -5393.441} C_VEL
LIN {X 0,Y 510.184,Z 668.989,A -85,B 0,C 180,E1 -5394.466,E2 -5394.466} C_VEL
LIN {X 0,Y 510.541,Z 658.31,A -85,B 0,C 180,E1 -5395.46,E2 -5395.46} C_VEL
LIN {X 0,Y 510.873,Z 647.607,A -85,B 0,C 180,E1 -5396.253,E2 -5396.253} C_VEL
LIN {X 0,Y 511.115,Z 637.623,A -85,B 0,C 180,E1 -5396.847,E2 -5396.847} C_VEL
LIN {X 0,Y 511.392,Z 624.484,A -85,B 0,C 180,E1 -5397.44,E2 -5397.44} C_VEL
LIN {X 0,Y 511.642,Z 611.991,A -85,B 0,C 180,E1 -5397.835,E2 -5397.835} C_VEL
LIN {X 0,Y 511.749,Z 599.253,A -85,B 0,C 180,E1 -5398.081,E2 -5398.081} C_VEL
LIN {X 0,Y 512.212,Z 510.607,A -85,B 0,C 180,E1 -5399.373,E2 -5399.373} C_VEL
LIN {X 0,Y 510.261,Z 501.322,A -85,B 0,C 180,E1 -5399.581,E2 -5399.581} C_VEL
LIN {X 0,Y 510.069,Z 496.097,A -85,B 0,C 180,E1 -5400.839,E2 -5400.839} C_VEL
LIN {X 0,Y 509.952,Z 495.967,A -85,B 0,C 180,E1 -5403.16,E2 -5403.16} C_VEL
LIN {X 0,Y 509.974,Z 495.958,A -85,B 0,C 180,E1 -5406.33,E2 -5406.33} C_VEL
LIN {X 0,Y 509.91,Z 495.967,A -85,B 0,C 180,E1 -5408.72,E2 -5408.72} C_VEL
LIN {X 0,Y 509.941,Z 495.962,A -85,B 0,C 180,E1 -5411.931,E2 -5411.931} C_VEL
LIN {X 0,Y 509.884,Z 495.975,A -85,B 0,C 180,E1 -5415.242,E2 -5415.242} C_VEL
LIN {X 0,Y 509.879,Z 495.968,A -85,B 0,C 180,E1 -5418.001,E2 -5418.001} C_VEL
LIN {X 0,Y 509.842,Z 495.979,A -85,B 0,C 180,E1 -5421.002,E2 -5421.002} C_VEL
LIN {X 0,Y 509.828,Z 495.977,A -85,B 0,C 180,E1 -5423.564,E2 -5423.564} C_VEL
LIN {X 0,Y 509.905,Z 495.964,A -85,B 0,C 180,E1 -5426.38,E2 -5426.38} C_VEL
LIN {X 0,Y 509.878,Z 495.972,A -85,B 0,C 180,E1 -5428.844,E2 -5428.844} C_VEL
LIN {X 0,Y 509.819,Z 495.976,A -85,B 0,C 180,E1 -5431.59,E2 -5431.59} C_VEL
LIN {X 0,Y 509.848,Z 495.971,A -85,B 0,C 180,E1 -5434.414,E2 -5434.414} C_VEL
LIN {X 0,Y 509.813,Z 495.98,A -85,B 0,C 180,E1 -5437.341,E2 -5437.341} C_VEL
LIN {X 0,Y 509.833,Z 495.975,A -85,B 0,C 180,E1 -5440.383,E2 -5440.383} C_VEL
LIN {X 0,Y 509.819,Z 495.983,A -85,B 0,C 180,E1 -5443.063,E2 -5443.063} C_VEL
LIN {X 0,Y 509.826,Z 495.976,A -85,B 0,C 180,E1 -5445.793,E2 -5445.793} C_VEL
LIN {X 0,Y 509.855,Z 495.976,A -85,B 0,C 180,E1 -5448.576,E2 -5448.576} C_VEL
LIN {X 0,Y 509.849,Z 495.973,A -85,B 0,C 180,E1 -5451.787,E2 -5451.787} C_VEL
LIN {X 0,Y 509.84,Z 495.979,A -85,B 0,C 180,E1 -5454.624,E2 -5454.624} C_VEL
LIN {X 0,Y 509.864,Z 495.975,A -85,B 0,C 180,E1 -5457.482,E2 -5457.482} C_VEL
LIN {X 0,Y 509.857,Z 495.977,A -85,B 0,C 180,E1 -5460.274,E2 -5460.274} C_VEL
LIN {X 0,Y 509.886,Z 495.975,A -85,B 0,C 180,E1 -5462.945,E2 -5462.945} C_VEL
LIN {X 0,Y 509.929,Z 496.191,A -85,B 0,C 180,E1 -5463.469,E2 -5463.469} C_VEL
LIN {X 0,Y 511.961,Z 506.716,A -85,B 0,C 180,E1 -5465.116,E2 -5465.116} C_VEL
LIN {X 0,Y 511.436,Z 526.891,A -85,B 0,C 180,E1 -5468.01,E2 -5468.01} C_VEL
LIN {X 0,Y 510.865,Z 549.079,A -85,B 0,C 180,E1 -5471.138,E2 -5471.138} C_VEL
LIN {X 0,Y 510.383,Z 572.584,A -85,B 0,C 180,E1 -5474.406,E2 -5474.406} C_VEL
LIN {X 0,Y 512.17,Z 587.141,A -85,B 0,C 180,E1 -5474.694,E2 -5474.694} C_VEL
LIN {X 0,Y 511.658,Z 682.054,A -85,B 0,C 180,E1 -5476.066,E2 -5476.066} C_VEL
LIN {X 0,Y 511.349,Z 695.363,A -85,B 0,C 180,E1 -5476.412,E2 -5476.412} C_VEL
LIN {X 0,Y 511.084,Z 708.757,A -85,B 0,C 180,E1 -5476.937,E2 -5476.937} C_VEL
LIN {X 0,Y 510.781,Z 721.236,A -85,B 0,C 180,E1 -5477.611,E2 -5477.611} C_VEL
LIN {X 0,Y 510.454,Z 732.398,A -85,B 0,C 180,E1 -5478.384,E2 -5478.384} C_VEL
LIN {X 0,Y 510.127,Z 742.827,A -85,B 0,C 180,E1 -5479.281,E2 -5479.281} C_VEL
LIN {X 0,Y 509.855,Z 752.234,A -85,B 0,C 180,E1 -5480.279,E2 -5480.279} C_VEL
LIN {X 0,Y 509.63,Z 761.355,A -85,B 0,C 180,E1 -5481.475,E2 -5481.475} C_VEL
LIN {X 0,Y 509.436,Z 768.671,A -85,B 0,C 180,E1 -5482.669,E2 -5482.669} C_VEL
LIN {X 0,Y 509.368,Z 775.376,A -85,B 0,C 180,E1 -5484.06,E2 -5484.06} C_VEL
LIN {X 0,Y 509.188,Z 779.793,A -85,B 0,C 180,E1 -5485.25,E2 -5485.25} C_VEL
LIN {X 0,Y 509.283,Z 782.13,A -85,B 0,C 180,E1 -5486.044,E2 -5486.044} C_VEL
LIN {X 0,Y 509.2,Z 784.018,A -85,B 0,C 180,E1 -5486.835,E2 -5486.835} C_VEL
LIN {X 0,Y 509.189,Z 785.452,A -85,B 0,C 180,E1 -5487.627,E2 -5487.627} C_VEL
LIN {X 0,Y 509.08,Z 787.084,A -85,B 0,C 180,E1 -5489.209,E2 -5489.209} C_VEL
LIN {X 0,Y 509.075,Z 787.302,A -85,B 0,C 180,E1 -5490,E2 -5490} C_VEL
LIN {X 0,Y 509.08,Z 787.089,A -85,B 0,C 180,E1 -5490.791,E2 -5490.791} C_VEL
LIN {X 0,Y 509.189,Z 785.479,A -85,B 0,C 180,E1 -5492.373,E2 -5492.373} C_VEL
LIN {X 0,Y 509.2,Z 784.053,A -85,B 0,C 180,E1 -5493.165,E2 -5493.165} C_VEL
LIN {X 0,Y 509.238,Z 781.091,A -85,B 0,C 180,E1 -5494.353,E2 -5494.353} C_VEL
LIN {X 0,Y 509.344,Z 777.069,A -85,B 0,C 180,E1 -5495.543,E2 -5495.543} C_VEL
LIN {X 0,Y 509.395,Z 771.33,A -85,B 0,C 180,E1 -5496.844,E2 -5496.844} C_VEL
LIN {X 0,Y 509.537,Z 764.102,A -85,B 0,C 180,E1 -5498.127,E2 -5498.127} C_VEL
LIN {X 0,Y 509.775,Z 755.692,A -85,B 0,C 180,E1 -5499.322,E2 -5499.322} C_VEL
LIN {X 0,Y 510.016,Z 747.044,A -85,B 0,C 180,E1 -5500.319,E2 -5500.319} C_VEL
LIN {X 0,Y 510.418,Z 736.433,A -85,B 0,C 180,E1 -5501.315,E2 -5501.315} C_VEL
LIN {X 0,Y 510.67,Z 725.688,A -85,B 0,C 180,E1 -5502.127,E2 -5502.127} C_VEL
LIN {X 0,Y 510.962,Z 714.266,A -85,B 0,C 180,E1 -5502.814,E2 -5502.814} C_VEL
LIN {X 0,Y 511.253,Z 702.246,A -85,B 0,C 180,E1 -5503.362,E2 -5503.362} C_VEL
LIN {X 0,Y 511.547,Z 689.271,A -85,B 0,C 180,E1 -5503.785,E2 -5503.785} C_VEL
LIN {X 0,Y 511.72,Z 675.585,A -85,B 0,C 180,E1 -5504.059,E2 -5504.059} C_VEL
LIN {X 0,Y 512.139,Z 585.676,A -85,B 0,C 180,E1 -5505.339,E2 -5505.339} C_VEL
LIN {X 0,Y 510.442,Z 573.24,A -85,B 0,C 180,E1 -5505.601,E2 -5505.601} C_VEL
LIN {X 0,Y 511.038,Z 548.716,A -85,B 0,C 180,E1 -5509.063,E2 -5509.063} C_VEL
LIN {X 0,Y 511.605,Z 526.663,A -85,B 0,C 180,E1 -5512.195,E2 -5512.195} C_VEL
LIN {X 0,Y 512.195,Z 509.287,A -85,B 0,C 180,E1 -5514.71,E2 -5514.71} C_VEL
LIN {X 0,Y 511.708,Z 504.678,A -85,B 0,C 180,E1 -5515.416,E2 -5515.416} C_VEL
LIN {X 0,Y 509.909,Z 495.971,A -85,B 0,C 180,E1 -5516.836,E2 -5516.836} C_VEL
LIN {X 0,Y 509.856,Z 495.974,A -85,B 0,C 180,E1 -5519.75,E2 -5519.75} C_VEL
LIN {X 0,Y 509.873,Z 495.973,A -85,B 0,C 180,E1 -5522.774,E2 -5522.774} C_VEL
LIN {X 0,Y 509.824,Z 495.977,A -85,B 0,C 180,E1 -5525.578,E2 -5525.578} C_VEL
LIN {X 0,Y 509.847,Z 495.959,A -85,B 0,C 180,E1 -5528.337,E2 -5528.337} C_VEL
LIN {X 0,Y 509.855,Z 495.977,A -85,B 0,C 180,E1 -5531.424,E2 -5531.424} C_VEL
LIN {X 0,Y 509.852,Z 495.971,A -85,B 0,C 180,E1 -5534.667,E2 -5534.667} C_VEL
LIN {X 0,Y 509.856,Z 495.967,A -85,B 0,C 180,E1 -5538.102,E2 -5538.102} C_VEL
LIN {X 0,Y 509.842,Z 495.974,A -85,B 0,C 180,E1 -5540.647,E2 -5540.647} C_VEL
LIN {X 0,Y 509.829,Z 495.973,A -85,B 0,C 180,E1 -5543.647,E2 -5543.647} C_VEL
LIN {X 0,Y 509.857,Z 495.972,A -85,B 0,C 180,E1 -5546.539,E2 -5546.539} C_VEL
LIN {X 0,Y 509.843,Z 495.974,A -85,B 0,C 180,E1 -5549.334,E2 -5549.334} C_VEL
LIN {X 0,Y 509.887,Z 495.966,A -85,B 0,C 180,E1 -5552.054,E2 -5552.054} C_VEL
LIN {X 0,Y 509.869,Z 495.97,A -85,B 0,C 180,E1 -5554.704,E2 -5554.704} C_VEL
LIN {X 0,Y 509.847,Z 495.974,A -85,B 0,C 180,E1 -5557.449,E2 -5557.449} C_VEL
LIN {X 0,Y 509.908,Z 495.964,A -85,B 0,C 180,E1 -5559.844,E2 -5559.844} C_VEL
LIN {X 0,Y 509.877,Z 495.967,A -85,B 0,C 180,E1 -5563.175,E2 -5563.175} C_VEL
LIN {X 0,Y 509.854,Z 495.972,A -85,B 0,C 180,E1 -5565.634,E2 -5565.634} C_VEL
LIN {X 0,Y 509.919,Z 495.968,A -85,B 0,C 180,E1 -5568.875,E2 -5568.875} C_VEL
LIN {X 0,Y 509.942,Z 495.951,A -85,B 0,C 180,E1 -5572.078,E2 -5572.078} C_VEL
LIN {X 0,Y 510.001,Z 495.952,A -85,B 0,C 180,E1 -5574.465,E2 -5574.465} C_VEL
LIN {X 0,Y 510.046,Z 495.946,A -85,B 0,C 180,E1 -5577.631,E2 -5577.631} C_VEL
LIN {X 0,Y 510.057,Z 495.94,A -85,B 0,C 180,E1 -5580.79,E2 -5580.79} C_VEL
LIN {X 0,Y 509.953,Z 495.966,A -85,B 0,C 180,E1 -5583.16,E2 -5583.16} C_VEL
LIN {X 0,Y 509.974,Z 495.954,A -85,B 0,C 180,E1 -5586.33,E2 -5586.33} C_VEL
LIN {X 0,Y 509.91,Z 495.959,A -85,B 0,C 180,E1 -5588.721,E2 -5588.721} C_VEL
LIN {X 0,Y 509.896,Z 495.965,A -85,B 0,C 180,E1 -5591.932,E2 -5591.932} C_VEL
LIN {X 0,Y 509.884,Z 495.965,A -85,B 0,C 180,E1 -5595.242,E2 -5595.242} C_VEL
LIN {X 0,Y 509.88,Z 495.965,A -85,B 0,C 180,E1 -5598.002,E2 -5598.002} C_VEL
LIN {X 0,Y 509.843,Z 495.98,A -85,B 0,C 180,E1 -5601.002,E2 -5601.002} C_VEL
LIN {X 0,Y 509.829,Z 495.972,A -85,B 0,C 180,E1 -5603.564,E2 -5603.564} C_VEL
LIN {X 0,Y 509.907,Z 495.965,A -85,B 0,C 180,E1 -5606.38,E2 -5606.38} C_VEL
LIN {X 0,Y 509.879,Z 495.972,A -85,B 0,C 180,E1 -5608.844,E2 -5608.844} C_VEL
LIN {X 0,Y 509.821,Z 495.977,A -85,B 0,C 180,E1 -5611.591,E2 -5611.591} C_VEL
LIN {X 0,Y 509.85,Z 495.971,A -85,B 0,C 180,E1 -5614.414,E2 -5614.414} C_VEL
LIN {X 0,Y 509.818,Z 495.981,A -85,B 0,C 180,E1 -5617.341,E2 -5617.341} C_VEL
LIN {X 0,Y 509.835,Z 495.974,A -85,B 0,C 180,E1 -5620.383,E2 -5620.383} C_VEL
LIN {X 0,Y 509.836,Z 495.98,A -85,B 0,C 180,E1 -5623.065,E2 -5623.065} C_VEL
LIN {X 0,Y 509.829,Z 495.975,A -85,B 0,C 180,E1 -5625.793,E2 -5625.793} C_VEL
LIN {X 0,Y 509.858,Z 495.974,A -85,B 0,C 180,E1 -5628.576,E2 -5628.576} C_VEL
LIN {X 0,Y 509.851,Z 495.971,A -85,B 0,C 180,E1 -5631.787,E2 -5631.787} C_VEL
LIN {X 0,Y 509.819,Z 495.976,A -85,B 0,C 180,E1 -5633.75,E2 -5633.75} C_VEL
LIN {X 0,Y 509.152,Z 496.061,A -85,B 0,C 180,E1 -5634.409,E2 -5634.409} C_VEL
LIN {X 0,Y 506.339,Z 496.415,A -85,B 0,C 180,E1 -5635.481,E2 -5635.481} C_VEL
LIN {X 0,Y 503.952,Z 496.715,A -85,B 0,C 180,E1 -5636.345,E2 -5636.345} C_VEL
LIN {X 0,Y 502.905,Z 496.843,A -85,B 0,C 180,E1 -5637.011,E2 -5637.011} C_VEL
LIN {X 0,Y 502.808,Z 496.851,A -85,B 0,C 180,E1 -5637.237,E2 -5637.237} C_VEL
LIN {X 0,Y 502.816,Z 496.849,A -85,B 0,C 180,E1 -5640.066,E2 -5640.066} C_VEL
LIN {X 0,Y 502.835,Z 496.849,A -85,B 0,C 180,E1 -5642.534,E2 -5642.534} C_VEL
LIN {X 0,Y 502.89,Z 497.001,A -85,B 0,C 180,E1 -5644.05,E2 -5644.05} C_VEL
LIN {X 0,Y 504.32,Z 505.391,A -85,B 0,C 180,E1 -5645.508,E2 -5645.508} C_VEL
LIN {X 0,Y 504.059,Z 518.483,A -85,B 0,C 180,E1 -5647.671,E2 -5647.671} C_VEL
LIN {X 0,Y 503.63,Z 536.684,A -85,B 0,C 180,E1 -5650.645,E2 -5650.645} C_VEL
LIN {X 0,Y 503.444,Z 546.677,A -85,B 0,C 180,E1 -5652.246,E2 -5652.246} C_VEL
LIN {X 0,Y 505.445,Z 558.485,A -85,B 0,C 180,E1 -5652.487,E2 -5652.487} C_VEL
LIN {X 0,Y 504.856,Z 655.151,A -85,B 0,C 180,E1 -5653.886,E2 -5653.886} C_VEL
LIN {X 0,Y 504.69,Z 668.137,A -85,B 0,C 180,E1 -5654.231,E2 -5654.231} C_VEL
LIN {X 0,Y 504.401,Z 681.078,A -85,B 0,C 180,E1 -5654.753,E2 -5654.753} C_VEL
LIN {X 0,Y 504.07,Z 692.344,A -85,B 0,C 180,E1 -5655.363,E2 -5655.363} C_VEL
LIN {X 0,Y 503.631,Z 704.031,A -85,B 0,C 180,E1 -5656.174,E2 -5656.174} C_VEL
LIN {X 0,Y 503.281,Z 714.411,A -85,B 0,C 180,E1 -5657.09,E2 -5657.09} C_VEL
LIN {X 0,Y 502.942,Z 724.285,A -85,B 0,C 180,E1 -5658.164,E2 -5658.164} C_VEL
LIN {X 0,Y 502.726,Z 732.826,A -85,B 0,C 180,E1 -5659.326,E2 -5659.326} C_VEL
LIN {X 0,Y 502.456,Z 740.064,A -85,B 0,C 180,E1 -5660.541,E2 -5660.541} C_VEL
LIN {X 0,Y 502.286,Z 746.715,A -85,B 0,C 180,E1 -5661.957,E2 -5661.957} C_VEL
LIN {X 0,Y 502.209,Z 751.192,A -85,B 0,C 180,E1 -5663.209,E2 -5663.209} C_VEL
LIN {X 0,Y 502.16,Z 754.355,A -85,B 0,C 180,E1 -5664.378,E2 -5664.378} C_VEL
LIN {X 0,Y 502.086,Z 757.21,A -85,B 0,C 180,E1 -5665.987,E2 -5665.987} C_VEL
LIN {X 0,Y 502.107,Z 758.043,A -85,B 0,C 180,E1 -5666.791,E2 -5666.791} C_VEL
LIN {X 0,Y 502.09,Z 758.444,A -85,B 0,C 180,E1 -5667.593,E2 -5667.593} C_VEL
LIN {X 0,Y 501.991,Z 758.109,A -85,B 0,C 180,E1 -5669.198,E2 -5669.198} C_VEL
LIN {X 0,Y 501.983,Z 757.354,A -85,B 0,C 180,E1 -5670,E2 -5670} C_VEL
LIN {X 0,Y 502.067,Z 754.592,A -85,B 0,C 180,E1 -5671.604,E2 -5671.604} C_VEL
LIN {X 0,Y 502.21,Z 751.411,A -85,B 0,C 180,E1 -5672.807,E2 -5672.807} C_VEL
LIN {X 0,Y 502.298,Z 747.184,A -85,B 0,C 180,E1 -5674.012,E2 -5674.012} C_VEL
LIN {X 0,Y 502.501,Z 741.79,A -85,B 0,C 180,E1 -5675.216,E2 -5675.216} C_VEL
LIN {X 0,Y 502.669,Z 735.052,A -85,B 0,C 180,E1 -5676.422,E2 -5676.422} C_VEL
LIN {X 0,Y 502.891,Z 726.611,A -85,B 0,C 180,E1 -5677.629,E2 -5677.629} C_VEL
LIN {X 0,Y 503.175,Z 717.986,A -85,B 0,C 180,E1 -5678.635,E2 -5678.635} C_VEL
LIN {X 0,Y 503.638,Z 707.363,A -85,B 0,C 180,E1 -5679.64,E2 -5679.64} C_VEL
LIN {X 0,Y 503.923,Z 696.712,A -85,B 0,C 180,E1 -5680.446,E2 -5680.446} C_VEL
LIN {X 0,Y 504.297,Z 684.901,A -85,B 0,C 180,E1 -5681.149,E2 -5681.149} C_VEL
LIN {X 0,Y 504.604,Z 672.518,A -85,B 0,C 180,E1 -5681.702,E2 -5681.702} C_VEL
LIN {X 0,Y 504.78,Z 659.583,A -85,B 0,C 180,E1 -5682.105,E2 -5682.105} C_VEL
LIN {X 0,Y 504.991,Z 645.97,A -85,B 0,C 180,E1 -5682.355,E2 -5682.355} C_VEL
LIN {X 0,Y 505.366,Z 557.895,A -85,B 0,C 180,E1 -5683.614,E2 -5683.614} C_VEL
LIN {X 0,Y 503.434,Z 546.628,A -85,B 0,C 180,E1 -5683.857,E2 -5683.857} C_VEL
LIN {X 0,Y 503.791,Z 530.813,A -85,B 0,C 180,E1 -5686.409,E2 -5686.409} C_VEL
LIN {X 0,Y 504.217,Z 511.677,A -85,B 0,C 180,E1 -5689.543,E2 -5689.543} C_VEL
LIN {X 0,Y 504.345,Z 505.01,A -85,B 0,C 180,E1 -5690.646,E2 -5690.646} C_VEL
LIN {X 0,Y 502.828,Z 496.852,A -85,B 0,C 180,E1 -5692.063,E2 -5692.063} C_VEL
LIN {X 0,Y 502.83,Z 496.857,A -85,B 0,C 180,E1 -5694.79,E2 -5694.79} C_VEL
LIN {X 0,Y 502.835,Z 496.85,A -85,B 0,C 180,E1 -5697.466,E2 -5697.466} C_VEL
LIN {X 0,Y 502.811,Z 496.851,A -85,B 0,C 180,E1 -5700.21,E2 -5700.21} C_VEL
LIN {X 0,Y 502.833,Z 496.852,A -85,B 0,C 180,E1 -5703.03,E2 -5703.03} C_VEL
LIN {X 0,Y 502.773,Z 496.853,A -85,B 0,C 180,E1 -5705.95,E2 -5705.95} C_VEL
LIN {X 0,Y 502.802,Z 496.856,A -85,B 0,C 180,E1 -5708.975,E2 -5708.975} C_VEL
LIN {X 0,Y 502.828,Z 496.847,A -85,B 0,C 180,E1 -5712.135,E2 -5712.135} C_VEL
LIN {X 0,Y 502.798,Z 496.848,A -85,B 0,C 180,E1 -5715.467,E2 -5715.467} C_VEL
LIN {X 0,Y 502.827,Z 496.846,A -85,B 0,C 180,E1 -5717.863,E2 -5717.863} C_VEL
LIN {X 0,Y 502.799,Z 496.856,A -85,B 0,C 180,E1 -5721.023,E2 -5721.023} C_VEL
LIN {X 0,Y 502.781,Z 496.855,A -85,B 0,C 180,E1 -5724.166,E2 -5724.166} C_VEL
LIN {X 0,Y 502.908,Z 497.001,A -85,B 0,C 180,E1 -5727.393,E2 -5727.393} C_VEL
LIN {X 0,Y 503.2,Z 500.888,A -85,B 0,C 180,E1 -5728.276,E2 -5728.276} C_VEL
LIN {X 0,Y 505.454,Z 512.568,A -85,B 0,C 180,E1 -5728.529,E2 -5728.529} C_VEL
LIN {X 0,Y 504.79,Z 607.031,A -85,B 0,C 180,E1 -5729.948,E2 -5729.948} C_VEL
LIN {X 0,Y 504.588,Z 620.217,A -85,B 0,C 180,E1 -5730.309,E2 -5730.309} C_VEL
LIN {X 0,Y 504.376,Z 632.628,A -85,B 0,C 180,E1 -5730.811,E2 -5730.811} C_VEL
LIN {X 0,Y 504.037,Z 644.339,A -85,B 0,C 180,E1 -5731.452,E2 -5731.452} C_VEL
LIN {X 0,Y 503.689,Z 655.62,A -85,B 0,C 180,E1 -5732.245,E2 -5732.245} C_VEL
LIN {X 0,Y 503.386,Z 665.978,A -85,B 0,C 180,E1 -5733.156,E2 -5733.156} C_VEL
LIN {X 0,Y 503.034,Z 674.852,A -85,B 0,C 180,E1 -5734.112,E2 -5734.112} C_VEL
LIN {X 0,Y 502.743,Z 683.852,A -85,B 0,C 180,E1 -5735.317,E2 -5735.317} C_VEL
LIN {X 0,Y 502.51,Z 691.039,A -85,B 0,C 180,E1 -5736.509,E2 -5736.509} C_VEL
LIN {X 0,Y 502.378,Z 697.275,A -85,B 0,C 180,E1 -5737.807,E2 -5737.807} C_VEL
LIN {X 0,Y 502.259,Z 702.055,A -85,B 0,C 180,E1 -5739.095,E2 -5739.095} C_VEL
LIN {X 0,Y 502.152,Z 705.583,A -85,B 0,C 180,E1 -5740.373,E2 -5740.373} C_VEL
LIN {X 0,Y 502.055,Z 707.303,A -85,B 0,C 180,E1 -5741.218,E2 -5741.218} C_VEL
LIN {X 0,Y 502.049,Z 708.683,A -85,B 0,C 180,E1 -5742.154,E2 -5742.154} C_VEL
LIN {X 0,Y 502.035,Z 709.394,A -85,B 0,C 180,E1 -5742.903,E2 -5742.903} C_VEL
LIN {X 0,Y 502.02,Z 709.776,A -85,B 0,C 180,E1 -5743.74,E2 -5743.74} C_VEL
LIN {X 0,Y 502.062,Z 709.551,A -85,B 0,C 180,E1 -5744.985,E2 -5744.985} C_VEL
LIN {X 0,Y 502.054,Z 708.374,A -85,B 0,C 180,E1 -5746.233,E2 -5746.233} C_VEL
LIN {X 0,Y 502.119,Z 707.04,A -85,B 0,C 180,E1 -5747.059,E2 -5747.059} C_VEL
LIN {X 0,Y 502.216,Z 703.975,A -85,B 0,C 180,E1 -5748.394,E2 -5748.394} C_VEL
LIN {X 0,Y 502.304,Z 700.397,A -85,B 0,C 180,E1 -5749.52,E2 -5749.52} C_VEL
LIN {X 0,Y 502.453,Z 695.414,A -85,B 0,C 180,E1 -5750.743,E2 -5750.743} C_VEL
LIN {X 0,Y 502.623,Z 689.145,A -85,B 0,C 180,E1 -5751.962,E2 -5751.962} C_VEL
LIN {X 0,Y 502.875,Z 681.429,A -85,B 0,C 180,E1 -5753.157,E2 -5753.157} C_VEL
LIN {X 0,Y 503.105,Z 673.284,A -85,B 0,C 180,E1 -5754.187,E2 -5754.187} C_VEL
LIN {X 0,Y 503.452,Z 663.511,A -85,B 0,C 180,E1 -5755.195,E2 -5755.195} C_VEL
LIN {X 0,Y 503.736,Z 653.935,A -85,B 0,C 180,E1 -5756,E2 -5756} C_VEL
LIN {X 0,Y 504.021,Z 643.604,A -85,B 0,C 180,E1 -5756.702,E2 -5756.702} C_VEL
LIN {X 0,Y 504.39,Z 631.14,A -85,B 0,C 180,E1 -5757.354,E2 -5757.354} C_VEL
LIN {X 0,Y 504.629,Z 618.072,A -85,B 0,C 180,E1 -5757.855,E2 -5757.855} C_VEL
LIN {X 0,Y 504.819,Z 604.734,A -85,B 0,C 180,E1 -5758.18,E2 -5758.18} C_VEL
LIN {X 0,Y 505.419,Z 511.676,A -85,B 0,C 180,E1 -5759.573,E2 -5759.573} C_VEL
LIN {X 0,Y 503.336,Z 501.952,A -85,B 0,C 180,E1 -5759.805,E2 -5759.805} C_VEL
LIN {X 0,Y 503.174,Z 497.821,A -85,B 0,C 180,E1 -5760.8,E2 -5760.8} C_VEL
LIN {X 0,Y 502.946,Z 496.839,A -85,B 0,C 180,E1 -5761.101,E2 -5761.101} C_VEL
LIN {X 0,Y 502.895,Z 496.846,A -85,B 0,C 180,E1 -5763.204,E2 -5763.204} C_VEL
LIN {X 0,Y 502.922,Z 496.837,A -85,B 0,C 180,E1 -5766.419,E2 -5766.419} C_VEL
LIN {X 0,Y 502.868,Z 496.846,A -85,B 0,C 180,E1 -5768.843,E2 -5768.843} C_VEL
LIN {X 0,Y 502.884,Z 496.84,A -85,B 0,C 180,E1 -5772.101,E2 -5772.101} C_VEL
LIN {X 0,Y 502.839,Z 496.852,A -85,B 0,C 180,E1 -5775.4,E2 -5775.4} C_VEL
LIN {X 0,Y 502.837,Z 496.845,A -85,B 0,C 180,E1 -5778.123,E2 -5778.123} C_VEL
LIN {X 0,Y 502.819,Z 496.849,A -85,B 0,C 180,E1 -5780.537,E2 -5780.537} C_VEL
LIN {X 0,Y 502.788,Z 496.859,A -85,B 0,C 180,E1 -5783.041,E2 -5783.041} C_VEL
LIN {X 0,Y 502.833,Z 496.847,A -85,B 0,C 180,E1 -5785.676,E2 -5785.676} C_VEL
LIN {X 0,Y 502.835,Z 496.844,A -85,B 0,C 180,E1 -5788.373,E2 -5788.373} C_VEL
LIN {X 0,Y 502.79,Z 496.852,A -85,B 0,C 180,E1 -5791.5,E2 -5791.5} C_VEL
LIN {X 0,Y 502.801,Z 496.849,A -85,B 0,C 180,E1 -5794.446,E2 -5794.446} C_VEL
LIN {X 0,Y 502.775,Z 496.859,A -85,B 0,C 180,E1 -5797.179,E2 -5797.179} C_VEL
LIN {X 0,Y 502.783,Z 496.852,A -85,B 0,C 180,E1 -5800.016,E2 -5800.016} C_VEL
LIN {X 0,Y 502.797,Z 496.85,A -85,B 0,C 180,E1 -5802.2,E2 -5802.2} C_VEL
LIN {X 0,Y 502.796,Z 496.854,A -85,B 0,C 180,E1 -5805.469,E2 -5805.469} C_VEL
LIN {X 0,Y 502.826,Z 496.848,A -85,B 0,C 180,E1 -5807.865,E2 -5807.865} C_VEL
LIN {X 0,Y 502.8,Z 496.858,A -85,B 0,C 180,E1 -5811.025,E2 -5811.025} C_VEL
LIN {X 0,Y 502.78,Z 496.854,A -85,B 0,C 180,E1 -5814.169,E2 -5814.169} C_VEL
LIN {X 0,Y 502.831,Z 496.856,A -85,B 0,C 180,E1 -5816.994,E2 -5816.994} C_VEL
LIN {X 0,Y 502.814,Z 496.853,A -85,B 0,C 180,E1 -5820.066,E2 -5820.066} C_VEL
LIN {X 0,Y 502.855,Z 496.851,A -85,B 0,C 180,E1 -5823.171,E2 -5823.171} C_VEL
LIN {X 0,Y 502.907,Z 497.111,A -85,B 0,C 180,E1 -5823.286,E2 -5823.286} C_VEL
LIN {X 0,Y 505.03,Z 508.832,A -85,B 0,C 180,E1 -5825.141,E2 -5825.141} C_VEL
LIN {X 0,Y 504.395,Z 530.736,A -85,B 0,C 180,E1 -5828.332,E2 -5828.332} C_VEL
LIN {X 0,Y 503.817,Z 551.391,A -85,B 0,C 180,E1 -5831.287,E2 -5831.287} C_VEL
LIN {X 0,Y 503.348,Z 572.063,A -85,B 0,C 180,E1 -5834.199,E2 -5834.199} C_VEL
LIN {X 0,Y 505.294,Z 587.836,A -85,B 0,C 180,E1 -5834.502,E2 -5834.502} C_VEL
LIN {X 0,Y 504.728,Z 681.853,A -85,B 0,C 180,E1 -5835.897,E2 -5835.897} C_VEL
LIN {X 0,Y 504.393,Z 695.776,A -85,B 0,C 180,E1 -5836.273,E2 -5836.273} C_VEL
LIN {X 0,Y 504.077,Z 708.844,A -85,B 0,C 180,E1 -5836.803,E2 -5836.803} C_VEL
LIN {X 0,Y 503.751,Z 721.146,A -85,B 0,C 180,E1 -5837.486,E2 -5837.486} C_VEL
LIN {X 0,Y 503.4,Z 732.888,A -85,B 0,C 180,E1 -5838.321,E2 -5838.321} C_VEL
LIN {X 0,Y 503.055,Z 743.094,A -85,B 0,C 180,E1 -5839.231,E2 -5839.231} C_VEL
LIN {X 0,Y 502.734,Z 753.171,A -85,B 0,C 180,E1 -5840.343,E2 -5840.343} C_VEL
LIN {X 0,Y 502.526,Z 762.033,A -85,B 0,C 180,E1 -5841.556,E2 -5841.556} C_VEL
LIN {X 0,Y 502.347,Z 769.116,A -85,B 0,C 180,E1 -5842.767,E2 -5842.767} C_VEL
LIN {X 0,Y 502.26,Z 774.765,A -85,B 0,C 180,E1 -5843.976,E2 -5843.976} C_VEL
LIN {X 0,Y 502.111,Z 779.208,A -85,B 0,C 180,E1 -5845.183,E2 -5845.183} C_VEL
LIN {X 0,Y 502.212,Z 781.547,A -85,B 0,C 180,E1 -5845.988,E2 -5845.988} C_VEL
LIN {X 0,Y 502.122,Z 783.442,A -85,B 0,C 180,E1 -5846.791,E2 -5846.791} C_VEL
LIN {X 0,Y 502.12,Z 784.889,A -85,B 0,C 180,E1 -5847.594,E2 -5847.594} C_VEL
LIN {X 0,Y 502.001,Z 786.543,A -85,B 0,C 180,E1 -5849.198,E2 -5849.198} C_VEL
LIN {X 0,Y 501.996,Z 786.762,A -85,B 0,C 180,E1 -5850,E2 -5850} C_VEL
LIN {X 0,Y 502,Z 786.553,A -85,B 0,C 180,E1 -5850.802,E2 -5850.802} C_VEL
LIN {X 0,Y 502.12,Z 784.946,A -85,B 0,C 180,E1 -5852.406,E2 -5852.406} C_VEL
LIN {X 0,Y 502.122,Z 783.508,A -85,B 0,C 180,E1 -5853.209,E2 -5853.209} C_VEL
LIN {X 0,Y 502.135,Z 780.542,A -85,B 0,C 180,E1 -5854.415,E2 -5854.415} C_VEL
LIN {X 0,Y 502.259,Z 776.514,A -85,B 0,C 180,E1 -5855.621,E2 -5855.621} C_VEL
LIN {X 0,Y 502.33,Z 770.407,A -85,B 0,C 180,E1 -5857.011,E2 -5857.011} C_VEL
LIN {X 0,Y 502.483,Z 763.521,A -85,B 0,C 180,E1 -5858.242,E2 -5858.242} C_VEL
LIN {X 0,Y 502.724,Z 755.076,A -85,B 0,C 180,E1 -5859.454,E2 -5859.454} C_VEL
LIN {X 0,Y 502.981,Z 746.398,A -85,B 0,C 180,E1 -5860.465,E2 -5860.465} C_VEL
LIN {X 0,Y 503.34,Z 736.955,A -85,B 0,C 180,E1 -5861.374,E2 -5861.374} C_VEL
LIN {X 0,Y 503.675,Z 724.888,A -85,B 0,C 180,E1 -5862.305,E2 -5862.305} C_VEL
LIN {X 0,Y 504.003,Z 713.499,A -85,B 0,C 180,E1 -5862.994,E2 -5862.994} C_VEL
LIN {X 0,Y 504.312,Z 701.395,A -85,B 0,C 180,E1 -5863.55,E2 -5863.55} C_VEL
LIN {X 0,Y 504.62,Z 688.308,A -85,B 0,C 180,E1 -5863.978,E2 -5863.978} C_VEL
LIN {X 0,Y 504.801,Z 675.956,A -85,B 0,C 180,E1 -5864.23,E2 -5864.23} C_VEL
LIN {X 0,Y 505.18,Z 585.598,A -85,B 0,C 180,E1 -5865.549,E2 -5865.549} C_VEL
LIN {X 0,Y 503.448,Z 572.801,A -85,B 0,C 180,E1 -5865.818,E2 -5865.818} C_VEL
LIN {X 0,Y 504.076,Z 548.251,A -85,B 0,C 180,E1 -5869.337,E2 -5869.337} C_VEL
LIN {X 0,Y 504.667,Z 527.714,A -85,B 0,C 180,E1 -5872.301,E2 -5872.301} C_VEL
LIN {X 0,Y 505.29,Z 509.713,A -85,B 0,C 180,E1 -5874.951,E2 -5874.951} C_VEL
LIN {X 0,Y 503.464,Z 499.81,A -85,B 0,C 180,E1 -5876.531,E2 -5876.531} C_VEL
LIN {X 0,Y 502.863,Z 496.849,A -85,B 0,C 180,E1 -5877.014,E2 -5877.014} C_VEL
LIN {X 0,Y 502.809,Z 496.851,A -85,B 0,C 180,E1 -5880.21,E2 -5880.21} C_VEL
LIN {X 0,Y 502.83,Z 496.853,A -85,B 0,C 180,E1 -5883.03,E2 -5883.03} C_VEL
LIN {X 0,Y 502.771,Z 496.852,A -85,B 0,C 180,E1 -5885.95,E2 -5885.95} C_VEL
LIN {X 0,Y 502.799,Z 496.842,A -85,B 0,C 180,E1 -5888.975,E2 -5888.975} C_VEL
LIN {X 0,Y 502.826,Z 496.847,A -85,B 0,C 180,E1 -5892.135,E2 -5892.135} C_VEL
LIN {X 0,Y 502.796,Z 496.856,A -85,B 0,C 180,E1 -5895.467,E2 -5895.467} C_VEL
LIN {X 0,Y 502.821,Z 496.849,A -85,B 0,C 180,E1 -5899.003,E2 -5899.003} C_VEL
LIN {X 0,Y 502.788,Z 496.85,A -85,B 0,C 180,E1 -5902.045,E2 -5902.045} C_VEL
LIN {X 0,Y 502.804,Z 496.853,A -85,B 0,C 180,E1 -5905.035,E2 -5905.035} C_VEL
LIN {X 0,Y 502.781,Z 496.849,A -85,B 0,C 180,E1 -5907.915,E2 -5907.915} C_VEL
LIN {X 0,Y 502.831,Z 496.844,A -85,B 0,C 180,E1 -5910.713,E2 -5910.713} C_VEL
LIN {X 0,Y 502.873,Z 496.843,A -85,B 0,C 180,E1 -5913.434,E2 -5913.434} C_VEL
LIN {X 0,Y 502.783,Z 496.843,A -85,B 0,C 180,E1 -5916.086,E2 -5916.086} C_VEL
LIN {X 0,Y 502.775,Z 496.854,A -85,B 0,C 180,E1 -5918.689,E2 -5918.689} C_VEL
LIN {X 0,Y 502.822,Z 496.85,A -85,B 0,C 180,E1 -5921.248,E2 -5921.248} C_VEL
LIN {X 0,Y 502.814,Z 496.841,A -85,B 0,C 180,E1 -5923.767,E2 -5923.767} C_VEL
LIN {X 0,Y 502.821,Z 496.846,A -85,B 0,C 180,E1 -5926.255,E2 -5926.255} C_VEL
LIN {X 0,Y 502.887,Z 496.842,A -85,B 0,C 180,E1 -5928.717,E2 -5928.717} C_VEL
LIN {X 0,Y 502.892,Z 496.829,A -85,B 0,C 180,E1 -5931.967,E2 -5931.967} C_VEL
LIN {X 0,Y 502.953,Z 496.829,A -85,B 0,C 180,E1 -5934.387,E2 -5934.387} C_VEL
LIN {X 0,Y 503.016,Z 496.822,A -85,B 0,C 180,E1 -5937.598,E2 -5937.598} C_VEL
LIN {X 0,Y 503.017,Z 496.812,A -85,B 0,C 180,E1 -5940,E2 -5940} C_VEL
LIN {X 0,Y 503.016,Z 496.82,A -85,B 0,C 180,E1 -5942.402,E2 -5942.402} C_VEL
LIN {X 0,Y 502.954,Z 496.83,A -85,B 0,C 180,E1 -5945.614,E2 -5945.614} C_VEL
LIN {X 0,Y 502.893,Z 496.829,A -85,B 0,C 180,E1 -5948.034,E2 -5948.034} C_VEL
LIN {X 0,Y 502.872,Z 496.846,A -85,B 0,C 180,E1 -5951.284,E2 -5951.284} C_VEL
LIN {X 0,Y 502.836,Z 496.845,A -85,B 0,C 180,E1 -5954.571,E2 -5954.571} C_VEL
LIN {X 0,Y 502.854,Z 496.841,A -85,B 0,C 180,E1 -5957.908,E2 -5957.908} C_VEL
LIN {X 0,Y 502.82,Z 496.849,A -85,B 0,C 180,E1 -5960.537,E2 -5960.537} C_VEL
LIN {X 0,Y 502.789,Z 496.852,A -85,B 0,C 180,E1 -5963.041,E2 -5963.041} C_VEL
LIN {X 0,Y 502.835,Z 496.846,A -85,B 0,C 180,E1 -5965.676,E2 -5965.676} C_VEL
LIN {X 0,Y 502.836,Z 496.844,A -85,B 0,C 180,E1 -5968.373,E2 -5968.373} C_VEL
LIN {X 0,Y 502.791,Z 496.853,A -85,B 0,C 180,E1 -5971.501,E2 -5971.501} C_VEL
LIN {X 0,Y 502.802,Z 496.849,A -85,B 0,C 180,E1 -5974.446,E2 -5974.446} C_VEL
LIN {X 0,Y 502.78,Z 496.86,A -85,B 0,C 180,E1 -5977.18,E2 -5977.18} C_VEL
LIN {X 0,Y 502.785,Z 496.851,A -85,B 0,C 180,E1 -5980.016,E2 -5980.016} C_VEL
LIN {X 0,Y 502.799,Z 496.852,A -85,B 0,C 180,E1 -5982.2,E2 -5982.2} C_VEL
LIN {X 0,Y 502.798,Z 496.853,A -85,B 0,C 180,E1 -5985.469,E2 -5985.469} C_VEL
LIN {X 0,Y 502.828,Z 496.847,A -85,B 0,C 180,E1 -5987.865,E2 -5987.865} C_VEL
LIN {X 0,Y 502.802,Z 496.857,A -85,B 0,C 180,E1 -5991.025,E2 -5991.025} C_VEL
LIN {X 0,Y 502.775,Z 496.853,A -85,B 0,C 180,E1 -5994.17,E2 -5994.17} C_VEL
LIN {X 0,Y 502.808,Z 496.851,A -85,B 0,C 180,E1 -5997.237,E2 -5997.237} C_VEL
LIN {X 0,Y 502.107,Z 496.936,A -85,B 0,C 180,E1 -5997.905,E2 -5997.905} C_VEL
LIN {X 0,Y 499.242,Z 497.3,A -85,B 0,C 180,E1 -5998.991,E2 -5998.991} C_VEL
LIN {X 0,Y 496.848,Z 497.595,A -85,B 0,C 180,E1 -5999.866,E2 -5999.866} C_VEL
LIN {X 0,Y 495.833,Z 497.721,A -85,B 0,C 180,E1 -6000.542,E2 -6000.542} C_VEL
LIN {X 0,Y 495.755,Z 497.73,A -85,B 0,C 180,E1 -6000.771,E2 -6000.771} C_VEL
LIN {X 0,Y 495.851,Z 497.919,A -85,B 0,C 180,E1 -6003.885,E2 -6003.885} C_VEL
LIN {X 0,Y 497.344,Z 506.328,A -85,B 0,C 180,E1 -6005.364,E2 -6005.364} C_VEL
LIN {X 0,Y 497.119,Z 519.469,A -85,B 0,C 180,E1 -6007.561,E2 -6007.561} C_VEL
LIN {X 0,Y 496.65,Z 537.782,A -85,B 0,C 180,E1 -6010.577,E2 -6010.577} C_VEL
LIN {X 0,Y 496.497,Z 546.715,A -85,B 0,C 180,E1 -6012.016,E2 -6012.016} C_VEL
LIN {X 0,Y 498.615,Z 559.677,A -85,B 0,C 180,E1 -6012.285,E2 -6012.285} C_VEL
LIN {X 0,Y 497.992,Z 655.521,A -85,B 0,C 180,E1 -6013.693,E2 -6013.693} C_VEL
LIN {X 0,Y 497.806,Z 668.548,A -85,B 0,C 180,E1 -6014.045,E2 -6014.045} C_VEL
LIN {X 0,Y 497.496,Z 681.708,A -85,B 0,C 180,E1 -6014.588,E2 -6014.588} C_VEL
LIN {X 0,Y 497.1,Z 693.727,A -85,B 0,C 180,E1 -6015.257,E2 -6015.257} C_VEL
LIN {X 0,Y 496.648,Z 705.106,A -85,B 0,C 180,E1 -6016.08,E2 -6016.08} C_VEL
LIN {X 0,Y 496.283,Z 715.34,A -85,B 0,C 180,E1 -6017.009,E2 -6017.009} C_VEL
LIN {X 0,Y 495.927,Z 724.873,A -85,B 0,C 180,E1 -6018.073,E2 -6018.073} C_VEL
LIN {X 0,Y 495.716,Z 732.83,A -85,B 0,C 180,E1 -6019.173,E2 -6019.173} C_VEL
LIN {X 0,Y 495.414,Z 740.1,A -85,B 0,C 180,E1 -6020.405,E2 -6020.405} C_VEL
LIN {X 0,Y 495.217,Z 746.795,A -85,B 0,C 180,E1 -6021.841,E2 -6021.841} C_VEL
LIN {X 0,Y 495.148,Z 751.177,A -85,B 0,C 180,E1 -6023.071,E2 -6023.071} C_VEL
LIN {X 0,Y 495.074,Z 754.486,A -85,B 0,C 180,E1 -6024.297,E2 -6024.297} C_VEL
LIN {X 0,Y 494.986,Z 757.364,A -85,B 0,C 180,E1 -6025.929,E2 -6025.929} C_VEL
LIN {X 0,Y 495.026,Z 758.213,A -85,B 0,C 180,E1 -6026.745,E2 -6026.745} C_VEL
LIN {X 0,Y 494.963,Z 758.661,A -85,B 0,C 180,E1 -6028.373,E2 -6028.373} C_VEL
LIN {X 0,Y 494.901,Z 757.58,A -85,B 0,C 180,E1 -6030,E2 -6030} C_VEL
LIN {X 0,Y 494.992,Z 754.841,A -85,B 0,C 180,E1 -6031.627,E2 -6031.627} C_VEL
LIN {X 0,Y 495.143,Z 751.683,A -85,B 0,C 180,E1 -6032.847,E2 -6032.847} C_VEL
LIN {X 0,Y 495.236,Z 747.48,A -85,B 0,C 180,E1 -6034.069,E2 -6034.069} C_VEL
LIN {X 0,Y 495.448,Z 742.111,A -85,B 0,C 180,E1 -6035.29,E2 -6035.29} C_VEL
LIN {X 0,Y 495.645,Z 735.41,A -85,B 0,C 180,E1 -6036.513,E2 -6036.513} C_VEL
LIN {X 0,Y 495.865,Z 727.01,A -85,B 0,C 180,E1 -6037.738,E2 -6037.738} C_VEL
LIN {X 0,Y 496.17,Z 718.424,A -85,B 0,C 180,E1 -6038.758,E2 -6038.758} C_VEL
LIN {X 0,Y 496.67,Z 707.875,A -85,B 0,C 180,E1 -6039.776,E2 -6039.776} C_VEL
LIN {X 0,Y 496.974,Z 697.292,A -85,B 0,C 180,E1 -6040.593,E2 -6040.593} C_VEL
LIN {X 0,Y 497.369,Z 685.57,A -85,B 0,C 180,E1 -6041.306,E2 -6041.306} C_VEL
LIN {X 0,Y 497.707,Z 673.415,A -85,B 0,C 180,E1 -6041.866,E2 -6041.866} C_VEL
LIN {X 0,Y 497.903,Z 659.785,A -85,B 0,C 180,E1 -6042.301,E2 -6042.301} C_VEL
LIN {X 0,Y 498.113,Z 646.177,A -85,B 0,C 180,E1 -6042.554,E2 -6042.554} C_VEL
LIN {X 0,Y 498.521,Z 558.683,A -85,B 0,C 180,E1 -6043.823,E2 -6043.823} C_VEL
LIN {X 0,Y 496.478,Z 546.703,A -85,B 0,C 180,E1 -6044.081,E2 -6044.081} C_VEL
LIN {X 0,Y 496.83,Z 529.606,A -85,B 0,C 180,E1 -6046.857,E2 -6046.857} C_VEL
LIN {X 0,Y 497.335,Z 510.376,A -85,B 0,C 180,E1 -6050.04,E2 -6050.04} C_VEL
LIN {X 0,Y 497.212,Z 505.107,A -85,B 0,C 180,E1 -6050.928,E2 -6050.928} C_VEL
LIN {X 0,Y 495.78,Z 497.731,A -85,B 0,C 180,E1 -6052.229,E2 -6052.229} C_VEL
LIN {X 0,Y 495.791,Z 497.733,A -85,B 0,C 180,E1 -6055.166,E2 -6055.166} C_VEL
LIN {X 0,Y 495.783,Z 497.726,A -85,B 0,C 180,E1 -6057.89,E2 -6057.89} C_VEL
LIN {X 0,Y 495.754,Z 497.734,A -85,B 0,C 180,E1 -6060.686,E2 -6060.686} C_VEL
LIN {X 0,Y 495.76,Z 497.727,A -85,B 0,C 180,E1 -6063.563,E2 -6063.563} C_VEL
LIN {X 0,Y 495.728,Z 497.734,A -85,B 0,C 180,E1 -6066.543,E2 -6066.543} C_VEL
LIN {X 0,Y 495.757,Z 497.726,A -85,B 0,C 180,E1 -6069.637,E2 -6069.637} C_VEL
LIN {X 0,Y 495.763,Z 497.73,A -85,B 0,C 180,E1 -6072.509,E2 -6072.509} C_VEL
LIN {X 0,Y 495.747,Z 497.729,A -85,B 0,C 180,E1 -6075.138,E2 -6075.138} C_VEL
LIN {X 0,Y 495.774,Z 497.726,A -85,B 0,C 180,E1 -6078.22,E2 -6078.22} C_VEL
LIN {X 0,Y 495.748,Z 497.73,A -85,B 0,C 180,E1 -6081.408,E2 -6081.408} C_VEL
LIN {X 0,Y 495.753,Z 497.733,A -85,B 0,C 180,E1 -6084.462,E2 -6084.462} C_VEL
LIN {X 0,Y 495.842,Z 497.796,A -85,B 0,C 180,E1 -6087.247,E2 -6087.247} C_VEL
LIN {X 0,Y 496.223,Z 501.141,A -85,B 0,C 180,E1 -6088.038,E2 -6088.038} C_VEL
LIN {X 0,Y 498.63,Z 513.192,A -85,B 0,C 180,E1 -6088.32,E2 -6088.32} C_VEL
LIN {X 0,Y 497.898,Z 607.667,A -85,B 0,C 180,E1 -6089.766,E2 -6089.766} C_VEL
LIN {X 0,Y 497.655,Z 621.182,A -85,B 0,C 180,E1 -6090.144,E2 -6090.144} C_VEL
LIN {X 0,Y 497.459,Z 633.481,A -85,B 0,C 180,E1 -6090.655,E2 -6090.655} C_VEL
LIN {X 0,Y 497.116,Z 644.564,A -85,B 0,C 180,E1 -6091.27,E2 -6091.27} C_VEL
LIN {X 0,Y 496.753,Z 655.63,A -85,B 0,C 180,E1 -6092.053,E2 -6092.053} C_VEL
LIN {X 0,Y 496.432,Z 665.787,A -85,B 0,C 180,E1 -6092.948,E2 -6092.948} C_VEL
LIN {X 0,Y 496.079,Z 675.05,A -85,B 0,C 180,E1 -6093.948,E2 -6093.948} C_VEL
LIN {X 0,Y 495.76,Z 683.86,A -85,B 0,C 180,E1 -6095.129,E2 -6095.129} C_VEL
LIN {X 0,Y 495.485,Z 691.369,A -85,B 0,C 180,E1 -6096.378,E2 -6096.378} C_VEL
LIN {X 0,Y 495.374,Z 696.698,A -85,B 0,C 180,E1 -6097.477,E2 -6097.477} C_VEL
LIN {X 0,Y 495.224,Z 701.755,A -85,B 0,C 180,E1 -6098.784,E2 -6098.784} C_VEL
LIN {X 0,Y 495.107,Z 705.534,A -85,B 0,C 180,E1 -6100.082,E2 -6100.082} C_VEL
LIN {X 0,Y 495.003,Z 707.402,A -85,B 0,C 180,E1 -6100.94,E2 -6100.94} C_VEL
LIN {X 0,Y 495.009,Z 709.115,A -85,B 0,C 180,E1 -6102.031,E2 -6102.031} C_VEL
LIN {X 0,Y 494.946,Z 710.263,A -85,B 0,C 180,E1 -6103.501,E2 -6103.501} C_VEL
LIN {X 0,Y 494.98,Z 710.147,A -85,B 0,C 180,E1 -6104.901,E2 -6104.901} C_VEL
LIN {X 0,Y 494.983,Z 709.226,A -85,B 0,C 180,E1 -6106.032,E2 -6106.032} C_VEL
LIN {X 0,Y 495.041,Z 708,A -85,B 0,C 180,E1 -6106.87,E2 -6106.87} C_VEL
LIN {X 0,Y 495.154,Z 704.843,A -85,B 0,C 180,E1 -6108.331,E2 -6108.331} C_VEL
LIN {X 0,Y 495.298,Z 700.277,A -85,B 0,C 180,E1 -6109.783,E2 -6109.783} C_VEL
LIN {X 0,Y 495.448,Z 694.086,A -85,B 0,C 180,E1 -6111.228,E2 -6111.228} C_VEL
LIN {X 0,Y 495.727,Z 687.318,A -85,B 0,C 180,E1 -6112.464,E2 -6112.464} C_VEL
LIN {X 0,Y 496.005,Z 678.903,A -85,B 0,C 180,E1 -6113.695,E2 -6113.695} C_VEL
LIN {X 0,Y 496.242,Z 670.264,A -85,B 0,C 180,E1 -6114.718,E2 -6114.718} C_VEL
LIN {X 0,Y 496.628,Z 659.604,A -85,B 0,C 180,E1 -6115.739,E2 -6115.739} C_VEL
LIN {X 0,Y 497.016,Z 648.94,A -85,B 0,C 180,E1 -6116.554,E2 -6116.554} C_VEL
LIN {X 0,Y 497.284,Z 638.98,A -85,B 0,C 180,E1 -6117.165,E2 -6117.165} C_VEL
LIN {X 0,Y 497.57,Z 625.906,A -85,B 0,C 180,E1 -6117.774,E2 -6117.774} C_VEL
LIN {X 0,Y 497.87,Z 612.583,A -85,B 0,C 180,E1 -6118.205,E2 -6118.205} C_VEL
LIN {X 0,Y 497.974,Z 599.472,A -85,B 0,C 180,E1 -6118.458,E2 -6118.458} C_VEL
LIN {X 0,Y 498.562,Z 512.518,A -85,B 0,C 180,E1 -6119.785,E2 -6119.785} C_VEL
LIN {X 0,Y 496.397,Z 502.63,A -85,B 0,C 180,E1 -6120.025,E2 -6120.025} C_VEL
LIN {X 0,Y 496.251,Z 499.396,A -85,B 0,C 180,E1 -6120.811,E2 -6120.811} C_VEL
LIN {X 0,Y 495.884,Z 497.719,A -85,B 0,C 180,E1 -6121.269,E2 -6121.269} C_VEL
LIN {X 0,Y 495.84,Z 497.724,A -85,B 0,C 180,E1 -6123.25,E2 -6123.25} C_VEL
LIN {X 0,Y 495.873,Z 497.715,A -85,B 0,C 180,E1 -6126.51,E2 -6126.51} C_VEL
LIN {X 0,Y 495.837,Z 497.724,A -85,B 0,C 180,E1 -6128.97,E2 -6128.97} C_VEL
LIN {X 0,Y 495.843,Z 497.717,A -85,B 0,C 180,E1 -6132.275,E2 -6132.275} C_VEL
LIN {X 0,Y 495.798,Z 497.726,A -85,B 0,C 180,E1 -6135.624,E2 -6135.624} C_VEL
LIN {X 0,Y 495.797,Z 497.722,A -85,B 0,C 180,E1 -6138.248,E2 -6138.248} C_VEL
LIN {X 0,Y 495.765,Z 497.729,A -85,B 0,C 180,E1 -6140.757,E2 -6140.757} C_VEL
LIN {X 0,Y 495.744,Z 497.734,A -85,B 0,C 180,E1 -6143.387,E2 -6143.387} C_VEL
LIN {X 0,Y 495.791,Z 497.722,A -85,B 0,C 180,E1 -6146.068,E2 -6146.068} C_VEL
LIN {X 0,Y 495.773,Z 497.728,A -85,B 0,C 180,E1 -6148.815,E2 -6148.815} C_VEL
LIN {X 0,Y 495.752,Z 497.727,A -85,B 0,C 180,E1 -6151.727,E2 -6151.727} C_VEL
LIN {X 0,Y 495.77,Z 497.727,A -85,B 0,C 180,E1 -6154.696,E2 -6154.696} C_VEL
LIN {X 0,Y 495.725,Z 497.732,A -85,B 0,C 180,E1 -6157.562,E2 -6157.562} C_VEL
LIN {X 0,Y 495.761,Z 497.73,A -85,B 0,C 180,E1 -6160.7,E2 -6160.7} C_VEL
LIN {X 0,Y 495.729,Z 497.731,A -85,B 0,C 180,E1 -6164.002,E2 -6164.002} C_VEL
LIN {X 0,Y 495.73,Z 497.738,A -85,B 0,C 180,E1 -6167.119,E2 -6167.119} C_VEL
LIN {X 0,Y 495.756,Z 497.729,A -85,B 0,C 180,E1 -6169.954,E2 -6169.954} C_VEL
LIN {X 0,Y 495.728,Z 497.736,A -85,B 0,C 180,E1 -6172.554,E2 -6172.554} C_VEL
LIN {X 0,Y 495.781,Z 497.729,A -85,B 0,C 180,E1 -6175.458,E2 -6175.458} C_VEL
LIN {X 0,Y 495.757,Z 497.734,A -85,B 0,C 180,E1 -6178.365,E2 -6178.365} C_VEL
LIN {X 0,Y 495.787,Z 497.729,A -85,B 0,C 180,E1 -6181.507,E2 -6181.507} C_VEL
LIN {X 0,Y 495.84,Z 497.803,A -85,B 0,C 180,E1 -6183.049,E2 -6183.049} C_VEL
LIN {X 0,Y 498.077,Z 509.548,A -85,B 0,C 180,E1 -6184.957,E2 -6184.957} C_VEL
LIN {X 0,Y 497.508,Z 528.658,A -85,B 0,C 180,E1 -6187.798,E2 -6187.798} C_VEL
LIN {X 0,Y 496.822,Z 550.773,A -85,B 0,C 180,E1 -6191.013,E2 -6191.013} C_VEL
LIN {X 0,Y 496.322,Z 571.471,A -85,B 0,C 180,E1 -6193.97,E2 -6193.97} C_VEL
LIN {X 0,Y 498.441,Z 588.404,A -85,B 0,C 180,E1 -6194.302,E2 -6194.302} C_VEL
LIN {X 0,Y 497.795,Z 681.649,A -85,B 0,C 180,E1 -6195.722,E2 -6195.722} C_VEL
LIN {X 0,Y 497.452,Z 695.424,A -85,B 0,C 180,E1 -6196.103,E2 -6196.103} C_VEL
LIN {X 0,Y 497.093,Z 707.889,A -85,B 0,C 180,E1 -6196.614,E2 -6196.614} C_VEL
LIN {X 0,Y 496.758,Z 719.319,A -85,B 0,C 180,E1 -6197.245,E2 -6197.245} C_VEL
LIN {X 0,Y 496.467,Z 730.771,A -85,B 0,C 180,E1 -6198.052,E2 -6198.052} C_VEL
LIN {X 0,Y 496.086,Z 741.298,A -85,B 0,C 180,E1 -6198.974,E2 -6198.974} C_VEL
LIN {X 0,Y 495.764,Z 750.82,A -85,B 0,C 180,E1 -6200,E2 -6200} C_VEL
LIN {X 0,Y 495.478,Z 760.013,A -85,B 0,C 180,E1 -6201.229,E2 -6201.229} C_VEL
LIN {X 0,Y 495.285,Z 767.368,A -85,B 0,C 180,E1 -6202.458,E2 -6202.458} C_VEL
LIN {X 0,Y 495.157,Z 773.493,A -85,B 0,C 180,E1 -6203.726,E2 -6203.726} C_VEL
LIN {X 0,Y 495.039,Z 778.609,A -85,B 0,C 180,E1 -6205.114,E2 -6205.114} C_VEL
LIN {X 0,Y 495.12,Z 780.963,A -85,B 0,C 180,E1 -6205.93,E2 -6205.93} C_VEL
LIN {X 0,Y 495.047,Z 782.866,A -85,B 0,C 180,E1 -6206.745,E2 -6206.745} C_VEL
LIN {X 0,Y 495.053,Z 784.326,A -85,B 0,C 180,E1 -6207.559,E2 -6207.559} C_VEL
LIN {X 0,Y 494.963,Z 785.366,A -85,B 0,C 180,E1 -6208.373,E2 -6208.373} C_VEL
LIN {X 0,Y 494.921,Z 786.001,A -85,B 0,C 180,E1 -6209.186,E2 -6209.186} C_VEL
LIN {X 0,Y 494.918,Z 786.221,A -85,B 0,C 180,E1 -6210,E2 -6210} C_VEL
LIN {X 0,Y 494.92,Z 786.016,A -85,B 0,C 180,E1 -6210.814,E2 -6210.814} C_VEL
LIN {X 0,Y 494.963,Z 785.413,A -85,B 0,C 180,E1 -6211.627,E2 -6211.627} C_VEL
LIN {X 0,Y 495.053,Z 784.406,A -85,B 0,C 180,E1 -6212.441,E2 -6212.441} C_VEL
LIN {X 0,Y 495.047,Z 782.962,A -85,B 0,C 180,E1 -6213.255,E2 -6213.255} C_VEL
LIN {X 0,Y 495.037,Z 779.991,A -85,B 0,C 180,E1 -6214.478,E2 -6214.478} C_VEL
LIN {X 0,Y 495.161,Z 774.828,A -85,B 0,C 180,E1 -6215.988,E2 -6215.988} C_VEL
LIN {X 0,Y 495.271,Z 768.697,A -85,B 0,C 180,E1 -6217.337,E2 -6217.337} C_VEL
LIN {X 0,Y 495.461,Z 761.643,A -85,B 0,C 180,E1 -6218.565,E2 -6218.565} C_VEL
LIN {X 0,Y 495.695,Z 752.862,A -85,B 0,C 180,E1 -6219.796,E2 -6219.796} C_VEL
LIN {X 0,Y 495.993,Z 743.802,A -85,B 0,C 180,E1 -6220.821,E2 -6220.821} C_VEL
LIN {X 0,Y 496.388,Z 732.659,A -85,B 0,C 180,E1 -6221.846,E2 -6221.846} C_VEL
LIN {X 0,Y 496.782,Z 721.603,A -85,B 0,C 180,E1 -6222.651,E2 -6222.651} C_VEL
LIN {X 0,Y 497.165,Z 708.735,A -85,B 0,C 180,E1 -6223.384,E2 -6223.384} C_VEL
LIN {X 0,Y 497.475,Z 695.721,A -85,B 0,C 180,E1 -6223.922,E2 -6223.922} C_VEL
LIN {X 0,Y 497.845,Z 681.889,A -85,B 0,C 180,E1 -6224.302,E2 -6224.302} C_VEL
LIN {X 0,Y 498.33,Z 606.613,A -85,B 0,C 180,E1 -6225.438,E2 -6225.438} C_VEL
LIN {X 0,Y 498.362,Z 586.548,A -85,B 0,C 180,E1 -6225.745,E2 -6225.745} C_VEL
LIN {X 0,Y 496.427,Z 572.382,A -85,B 0,C 180,E1 -6226.039,E2 -6226.039} C_VEL
LIN {X 0,Y 497.068,Z 549.222,A -85,B 0,C 180,E1 -6229.406,E2 -6229.406} C_VEL
LIN {X 0,Y 497.732,Z 528.766,A -85,B 0,C 180,E1 -6232.41,E2 -6232.41} C_VEL
LIN {X 0,Y 498.377,Z 511.225,A -85,B 0,C 180,E1 -6235.027,E2 -6235.027} C_VEL
LIN {X 0,Y 496.786,Z 502.391,A -85,B 0,C 180,E1 -6236.453,E2 -6236.453} C_VEL
LIN {X 0,Y 495.81,Z 497.727,A -85,B 0,C 180,E1 -6237.259,E2 -6237.259} C_VEL
LIN {X 0,Y 495.764,Z 497.728,A -85,B 0,C 180,E1 -6240.147,E2 -6240.147} C_VEL
LIN {X 0,Y 495.791,Z 497.731,A -85,B 0,C 180,E1 -6243.244,E2 -6243.244} C_VEL
LIN {X 0,Y 495.717,Z 497.73,A -85,B 0,C 180,E1 -6246.088,E2 -6246.088} C_VEL
LIN {X 0,Y 495.761,Z 497.715,A -85,B 0,C 180,E1 -6248.768,E2 -6248.768} C_VEL
LIN {X 0,Y 495.774,Z 497.727,A -85,B 0,C 180,E1 -6251.778,E2 -6251.778} C_VEL
LIN {X 0,Y 495.744,Z 497.735,A -85,B 0,C 180,E1 -6255.139,E2 -6255.139} C_VEL
LIN {X 0,Y 495.755,Z 497.723,A -85,B 0,C 180,E1 -6258.219,E2 -6258.219} C_VEL
LIN {X 0,Y 495.758,Z 497.734,A -85,B 0,C 180,E1 -6261.231,E2 -6261.231} C_VEL
LIN {X 0,Y 495.751,Z 497.725,A -85,B 0,C 180,E1 -6264.463,E2 -6264.463} C_VEL
LIN {X 0,Y 495.762,Z 497.728,A -85,B 0,C 180,E1 -6267.405,E2 -6267.405} C_VEL
LIN {X 0,Y 495.774,Z 497.72,A -85,B 0,C 180,E1 -6270.254,E2 -6270.254} C_VEL
LIN {X 0,Y 495.826,Z 497.724,A -85,B 0,C 180,E1 -6273.248,E2 -6273.248} C_VEL
LIN {X 0,Y 495.743,Z 497.721,A -85,B 0,C 180,E1 -6275.725,E2 -6275.725} C_VEL
LIN {X 0,Y 495.738,Z 497.728,A -85,B 0,C 180,E1 -6278.371,E2 -6278.371} C_VEL
LIN {X 0,Y 495.776,Z 497.73,A -85,B 0,C 180,E1 -6280.971,E2 -6280.971} C_VEL
LIN {X 0,Y 495.771,Z 497.721,A -85,B 0,C 180,E1 -6283.53,E2 -6283.53} C_VEL
LIN {X 0,Y 495.784,Z 497.722,A -85,B 0,C 180,E1 -6286.055,E2 -6286.055} C_VEL
LIN {X 0,Y 495.861,Z 497.715,A -85,B 0,C 180,E1 -6288.555,E2 -6288.555} C_VEL
LIN {X 0,Y 495.864,Z 497.705,A -85,B 0,C 180,E1 -6291.852,E2 -6291.852} C_VEL
LIN {X 0,Y 495.907,Z 497.706,A -85,B 0,C 180,E1 -6294.307,E2 -6294.307} C_VEL
LIN {X 0,Y 495.985,Z 497.698,A -85,B 0,C 180,E1 -6297.564,E2 -6297.564} C_VEL
LIN {X 0,Y 495.988,Z 497.686,A -85,B 0,C 180,E1 -6300,E2 -6300} C_VEL
LIN {X 0,Y 495.985,Z 497.696,A -85,B 0,C 180,E1 -6302.437,E2 -6302.437} C_VEL
LIN {X 0,Y 495.908,Z 497.707,A -85,B 0,C 180,E1 -6305.694,E2 -6305.694} C_VEL
LIN {X 0,Y 495.865,Z 497.704,A -85,B 0,C 180,E1 -6308.148,E2 -6308.148} C_VEL
LIN {X 0,Y 495.846,Z 497.719,A -85,B 0,C 180,E1 -6311.446,E2 -6311.446} C_VEL
LIN {X 0,Y 495.781,Z 497.727,A -85,B 0,C 180,E1 -6314.783,E2 -6314.783} C_VEL
LIN {X 0,Y 495.78,Z 497.727,A -85,B 0,C 180,E1 -6317.319,E2 -6317.319} C_VEL
LIN {X 0,Y 495.771,Z 497.725,A -85,B 0,C 180,E1 -6319.891,E2 -6319.891} C_VEL
LIN {X 0,Y 495.75,Z 497.729,A -85,B 0,C 180,E1 -6322.861,E2 -6322.861} C_VEL
LIN {X 0,Y 495.792,Z 497.722,A -85,B 0,C 180,E1 -6326.068,E2 -6326.068} C_VEL
LIN {X 0,Y 495.774,Z 497.729,A -85,B 0,C 180,E1 -6328.815,E2 -6328.815} C_VEL
LIN {X 0,Y 495.754,Z 497.728,A -85,B 0,C 180,E1 -6331.727,E2 -6331.727} C_VEL
LIN {X 0,Y 495.772,Z 497.727,A -85,B 0,C 180,E1 -6334.696,E2 -6334.696} C_VEL
LIN {X 0,Y 495.73,Z 497.733,A -85,B 0,C 180,E1 -6337.562,E2 -6337.562} C_VEL
LIN {X 0,Y 495.763,Z 497.73,A -85,B 0,C 180,E1 -6340.701,E2 -6340.701} C_VEL
LIN {X 0,Y 495.733,Z 497.729,A -85,B 0,C 180,E1 -6344.002,E2 -6344.002} C_VEL
LIN {X 0,Y 495.756,Z 497.733,A -85,B 0,C 180,E1 -6347.121,E2 -6347.121} C_VEL
LIN {X 0,Y 495.758,Z 497.727,A -85,B 0,C 180,E1 -6349.954,E2 -6349.954} C_VEL
LIN {X 0,Y 495.728,Z 497.733,A -85,B 0,C 180,E1 -6352.554,E2 -6352.554} C_VEL
LIN {X 0,Y 495.778,Z 497.728,A -85,B 0,C 180,E1 -6355.458,E2 -6355.458} C_VEL
LIN {X 0,Y 495.756,Z 497.726,A -85,B 0,C 180,E1 -6358.365,E2 -6358.365} C_VEL
LIN {X 0,Y 495.755,Z 497.73,A -85,B 0,C 180,E1 -6360.771,E2 -6360.771} C_VEL
LIN {X 0,Y 495.092,Z 497.818,A -85,B 0,C 180,E1 -6361.223,E2 -6361.223} C_VEL
LIN {X 0,Y 492.275,Z 498.17,A -85,B 0,C 180,E1 -6361.933,E2 -6361.933} C_VEL
LIN {X 0,Y 489.451,Z 498.522,A -85,B 0,C 180,E1 -6362.649,E2 -6362.649} C_VEL
LIN {X 0,Y 488.796,Z 498.602,A -85,B 0,C 180,E1 -6363.111,E2 -6363.111} C_VEL
LIN {X 0,Y 488.801,Z 498.78,A -85,B 0,C 180,E1 -6363.704,E2 -6363.704} C_VEL
LIN {X 0,Y 490.395,Z 507.402,A -85,B 0,C 180,E1 -6365.237,E2 -6365.237} C_VEL
LIN {X 0,Y 490.218,Z 519.173,A -85,B 0,C 180,E1 -6367.227,E2 -6367.227} C_VEL
LIN {X 0,Y 489.7,Z 537.576,A -85,B 0,C 180,E1 -6370.29,E2 -6370.29} C_VEL
LIN {X 0,Y 489.546,Z 546.754,A -85,B 0,C 180,E1 -6371.779,E2 -6371.779} C_VEL
LIN {X 0,Y 491.806,Z 560.171,A -85,B 0,C 180,E1 -6372.067,E2 -6372.067} C_VEL
LIN {X 0,Y 491.128,Z 655.719,A -85,B 0,C 180,E1 -6373.49,E2 -6373.49} C_VEL
LIN {X 0,Y 490.925,Z 668.63,A -85,B 0,C 180,E1 -6373.843,E2 -6373.843} C_VEL
LIN {X 0,Y 490.598,Z 681.27,A -85,B 0,C 180,E1 -6374.366,E2 -6374.366} C_VEL
LIN {X 0,Y 490.191,Z 693.425,A -85,B 0,C 180,E1 -6375.045,E2 -6375.045} C_VEL
LIN {X 0,Y 489.718,Z 704.934,A -85,B 0,C 180,E1 -6375.879,E2 -6375.879} C_VEL
LIN {X 0,Y 489.333,Z 715.231,A -85,B 0,C 180,E1 -6376.821,E2 -6376.821} C_VEL
LIN {X 0,Y 489.013,Z 723.713,A -85,B 0,C 180,E1 -6377.767,E2 -6377.767} C_VEL
LIN {X 0,Y 488.739,Z 731.443,A -85,B 0,C 180,E1 -6378.806,E2 -6378.806} C_VEL
LIN {X 0,Y 488.373,Z 739.047,A -85,B 0,C 180,E1 -6380.056,E2 -6380.056} C_VEL
LIN {X 0,Y 488.209,Z 745.114,A -85,B 0,C 180,E1 -6381.306,E2 -6381.306} C_VEL
LIN {X 0,Y 488.11,Z 749.916,A -85,B 0,C 180,E1 -6382.555,E2 -6382.555} C_VEL
LIN {X 0,Y 488.042,Z 752.921,A -85,B 0,C 180,E1 -6383.533,E2 -6383.533} C_VEL
LIN {X 0,Y 487.915,Z 756.265,A -85,B 0,C 180,E1 -6385.042,E2 -6385.042} C_VEL
LIN {X 0,Y 487.948,Z 758.38,A -85,B 0,C 180,E1 -6386.697,E2 -6386.697} C_VEL
LIN {X 0,Y 487.907,Z 758.815,A -85,B 0,C 180,E1 -6387.523,E2 -6387.523} C_VEL
LIN {X 0,Y 487.891,Z 758.856,A -85,B 0,C 180,E1 -6388.349,E2 -6388.349} C_VEL
LIN {X 0,Y 487.822,Z 757.803,A -85,B 0,C 180,E1 -6390,E2 -6390} C_VEL
LIN {X 0,Y 487.921,Z 755.09,A -85,B 0,C 180,E1 -6391.651,E2 -6391.651} C_VEL
LIN {X 0,Y 488.078,Z 751.955,A -85,B 0,C 180,E1 -6392.889,E2 -6392.889} C_VEL
LIN {X 0,Y 488.178,Z 747.775,A -85,B 0,C 180,E1 -6394.128,E2 -6394.128} C_VEL
LIN {X 0,Y 488.377,Z 742.433,A -85,B 0,C 180,E1 -6395.367,E2 -6395.367} C_VEL
LIN {X 0,Y 488.618,Z 735.763,A -85,B 0,C 180,E1 -6396.607,E2 -6396.607} C_VEL
LIN {X 0,Y 488.861,Z 727.407,A -85,B 0,C 180,E1 -6397.849,E2 -6397.849} C_VEL
LIN {X 0,Y 489.18,Z 718.86,A -85,B 0,C 180,E1 -6398.884,E2 -6398.884} C_VEL
LIN {X 0,Y 489.697,Z 708.378,A -85,B 0,C 180,E1 -6399.917,E2 -6399.917} C_VEL
LIN {X 0,Y 490.024,Z 697.87,A -85,B 0,C 180,E1 -6400.745,E2 -6400.745} C_VEL
LIN {X 0,Y 490.446,Z 686.238,A -85,B 0,C 180,E1 -6401.468,E2 -6401.468} C_VEL
LIN {X 0,Y 490.813,Z 674.271,A -85,B 0,C 180,E1 -6402.035,E2 -6402.035} C_VEL
LIN {X 0,Y 491.023,Z 660.974,A -85,B 0,C 180,E1 -6402.476,E2 -6402.476} C_VEL
LIN {X 0,Y 491.23,Z 648.149,A -85,B 0,C 180,E1 -6402.733,E2 -6402.733} C_VEL
LIN {X 0,Y 491.7,Z 559.55,A -85,B 0,C 180,E1 -6404.035,E2 -6404.035} C_VEL
LIN {X 0,Y 489.522,Z 546.781,A -85,B 0,C 180,E1 -6404.312,E2 -6404.312} C_VEL
LIN {X 0,Y 489.943,Z 528.403,A -85,B 0,C 180,E1 -6407.316,E2 -6407.316} C_VEL
LIN {X 0,Y 490.492,Z 509.046,A -85,B 0,C 180,E1 -6410.551,E2 -6410.551} C_VEL
LIN {X 0,Y 489.466,Z 502.397,A -85,B 0,C 180,E1 -6411.717,E2 -6411.717} C_VEL
LIN {X 0,Y 488.737,Z 498.61,A -85,B 0,C 180,E1 -6412.399,E2 -6412.399} C_VEL
LIN {X 0,Y 488.75,Z 498.605,A -85,B 0,C 180,E1 -6415.555,E2 -6415.555} C_VEL
LIN {X 0,Y 488.746,Z 498.603,A -85,B 0,C 180,E1 -6418.328,E2 -6418.328} C_VEL
LIN {X 0,Y 488.696,Z 498.614,A -85,B 0,C 180,E1 -6421.179,E2 -6421.179} C_VEL
LIN {X 0,Y 488.732,Z 498.602,A -85,B 0,C 180,E1 -6424.112,E2 -6424.112} C_VEL
LIN {X 0,Y 488.679,Z 498.615,A -85,B 0,C 180,E1 -6427.158,E2 -6427.158} C_VEL
LIN {X 0,Y 488.717,Z 498.604,A -85,B 0,C 180,E1 -6430.344,E2 -6430.344} C_VEL
LIN {X 0,Y 488.715,Z 498.604,A -85,B 0,C 180,E1 -6433.65,E2 -6433.65} C_VEL
LIN {X 0,Y 488.714,Z 498.603,A -85,B 0,C 180,E1 -6436.348,E2 -6436.348} C_VEL
LIN {X 0,Y 488.729,Z 498.603,A -85,B 0,C 180,E1 -6439.676,E2 -6439.676} C_VEL
LIN {X 0,Y 488.68,Z 498.616,A -85,B 0,C 180,E1 -6442.841,E2 -6442.841} C_VEL
LIN {X 0,Y 488.734,Z 498.605,A -85,B 0,C 180,E1 -6445.887,E2 -6445.887} C_VEL
LIN {X 0,Y 488.811,Z 498.753,A -85,B 0,C 180,E1 -6447.128,E2 -6447.128} C_VEL
LIN {X 0,Y 489.29,Z 501.819,A -85,B 0,C 180,E1 -6447.829,E2 -6447.829} C_VEL
LIN {X 0,Y 491.81,Z 514.087,A -85,B 0,C 180,E1 -6448.11,E2 -6448.11} C_VEL
LIN {X 0,Y 491.008,Z 607.703,A -85,B 0,C 180,E1 -6449.565,E2 -6449.565} C_VEL
LIN {X 0,Y 490.762,Z 621.331,A -85,B 0,C 180,E1 -6449.948,E2 -6449.948} C_VEL
LIN {X 0,Y 490.538,Z 634.3,A -85,B 0,C 180,E1 -6450.495,E2 -6450.495} C_VEL
LIN {X 0,Y 490.143,Z 646.584,A -85,B 0,C 180,E1 -6451.202,E2 -6451.202} C_VEL
LIN {X 0,Y 489.723,Z 658.444,A -85,B 0,C 180,E1 -6452.082,E2 -6452.082} C_VEL
LIN {X 0,Y 489.388,Z 668.29,A -85,B 0,C 180,E1 -6453.004,E2 -6453.004} C_VEL
LIN {X 0,Y 489.018,Z 677.029,A -85,B 0,C 180,E1 -6454.002,E2 -6454.002} C_VEL
LIN {X 0,Y 488.724,Z 685.209,A -85,B 0,C 180,E1 -6455.142,E2 -6455.142} C_VEL
LIN {X 0,Y 488.467,Z 693.002,A -85,B 0,C 180,E1 -6456.49,E2 -6456.49} C_VEL
LIN {X 0,Y 488.317,Z 698.037,A -85,B 0,C 180,E1 -6457.579,E2 -6457.579} C_VEL
LIN {X 0,Y 488.168,Z 702.906,A -85,B 0,C 180,E1 -6458.905,E2 -6458.905} C_VEL
LIN {X 0,Y 488.01,Z 706.506,A -85,B 0,C 180,E1 -6460.218,E2 -6460.218} C_VEL
LIN {X 0,Y 487.928,Z 709.534,A -85,B 0,C 180,E1 -6461.92,E2 -6461.92} C_VEL
LIN {X 0,Y 487.869,Z 710.705,A -85,B 0,C 180,E1 -6463.255,E2 -6463.255} C_VEL
LIN {X 0,Y 487.915,Z 710.75,A -85,B 0,C 180,E1 -6464.808,E2 -6464.808} C_VEL
LIN {X 0,Y 487.928,Z 710.008,A -85,B 0,C 180,E1 -6465.826,E2 -6465.826} C_VEL
LIN {X 0,Y 487.956,Z 708.947,A -85,B 0,C 180,E1 -6466.676,E2 -6466.676} C_VEL
LIN {X 0,Y 488.076,Z 705.682,A -85,B 0,C 180,E1 -6468.275,E2 -6468.275} C_VEL
LIN {X 0,Y 488.21,Z 701.614,A -85,B 0,C 180,E1 -6469.633,E2 -6469.633} C_VEL
LIN {X 0,Y 488.372,Z 696.648,A -85,B 0,C 180,E1 -6470.892,E2 -6470.892} C_VEL
LIN {X 0,Y 488.588,Z 690.395,A -85,B 0,C 180,E1 -6472.146,E2 -6472.146} C_VEL
LIN {X 0,Y 488.909,Z 682.536,A -85,B 0,C 180,E1 -6473.396,E2 -6473.396} C_VEL
LIN {X 0,Y 489.124,Z 674.564,A -85,B 0,C 180,E1 -6474.434,E2 -6474.434} C_VEL
